Fanuc TP program (LS listing): ultrahose.ls

/PROG  ultrahose
/ATTR
COMMENT	= "19-03-20 09:29:25";
PROG_SIZE	= 0;
DEFAULT_GROUP	= 1, *, *, *, *;
/APPL
    ARC Welding Equipment: 1, *, *, *, *;
/MN
   1:  CALL HOME_ALL;
   1:  UFRAME_NUM = 1;
   1:  UTOOL_NUM = 3;
   1:  COL GUARD ADJUST 150;
   1:  PR[91] = PR[90];
   1:  PR[91,1] = PR[90,1] + -71.989;
   1:  PR[91,2] = PR[90,2] + -18.440;
   1:  PR[91,3] = PR[90,3] + 1.495;
   1:  PR[92] = PR[91];
   1:  PR[92,3] = PR[92,3] + 20;
   1:J PR[92] 10% FINE;
   1:L PR[91] R[100]mm/sec CNT100;
   1:  CALL LASER_DRAHT_START;
   1:  PR[91,1] = PR[90,1] + -66.281;
   1:  PR[91,2] = PR[90,2] + -16.361;
   1:L PR[91] R[100]mm/sec CNT100;
   1:  PR[91,1] = PR[90,1] + -66.063;
   1:  PR[91,2] = PR[90,2] + -16.303;
   1:L PR[91] R[100]mm/sec CNT100;
   1:  PR[91,1] = PR[90,1] + -66.021;
   1:  PR[91,2] = PR[90,2] + -16.273;
   1:L PR[91] R[100]mm/sec CNT100;
   1:  PR[91,1] = PR[90,1] + -61.333;
   1:  PR[91,2] = PR[90,2] + -12.339;
   1:L PR[91] R[100]mm/sec CNT100;
   1:  PR[91,1] = PR[90,1] + -61.289;
   1:  PR[91,2] = PR[90,2] + -12.295;
   1:L PR[91] R[100]mm/sec CNT100;
   1:  PR[91,1] = PR[90,1] + -61.252;
   1:  PR[91,2] = PR[90,2] + -12.242;
   1:L PR[91] R[100]mm/sec CNT100;
   1:  PR[91,1] = PR[90,1] + -58.200;
   1:  PR[91,2] = PR[90,2] + -6.959;
   1:L PR[91] R[100]mm/sec CNT100;
   1:  PR[91,1] = PR[90,1] + -57.138;
   1:  PR[91,2] = PR[90,2] + -0.935;
   1:L PR[91] R[100]mm/sec CNT100;
   1:  PR[91,1] = PR[90,1] + -57.094;
   1:  PR[91,2] = PR[90,2] + -0.772;
   1:L PR[91] R[100]mm/sec CNT100;
   1:  PR[91,1] = PR[90,1] + -58.150;
   1:  PR[91,2] = PR[90,2] + 5.213;
   1:L PR[91] R[100]mm/sec CNT100;
   1:  PR[91,1] = PR[90,1] + -58.165;
   1:  PR[91,2] = PR[90,2] + 5.381;
   1:L PR[91] R[100]mm/sec CNT100;
   1:  PR[91,1] = PR[90,1] + -61.202;
   1:  PR[91,2] = PR[90,2] + 10.640;
   1:L PR[91] R[100]mm/sec CNT100;
   1:  PR[91,1] = PR[90,1] + -61.273;
   1:  PR[91,2] = PR[90,2] + 10.794;
   1:L PR[91] R[100]mm/sec CNT100;
   1:  PR[91,1] = PR[90,1] + -65.925;
   1:  PR[91,2] = PR[90,2] + 14.697;
   1:L PR[91] R[100]mm/sec CNT100;
   1:  PR[91,1] = PR[90,1] + -66.045;
   1:  PR[91,2] = PR[90,2] + 14.817;
   1:L PR[91] R[100]mm/sec CNT100;
   1:  PR[91,1] = PR[90,1] + -71.753;
   1:  PR[91,2] = PR[90,2] + 16.895;
   1:L PR[91] R[100]mm/sec CNT100;
   1:  PR[91,1] = PR[90,1] + -71.906;
   1:  PR[91,2] = PR[90,2] + 16.966;
   1:L PR[91] R[100]mm/sec CNT100;
   1:  PR[91,1] = PR[90,1] + -77.984;
   1:L PR[91] R[100]mm/sec CNT100;
   1:  PR[91,1] = PR[90,1] + -78.152;
   1:  PR[91,2] = PR[90,2] + 16.981;
   1:L PR[91] R[100]mm/sec CNT100;
   1:  PR[91,1] = PR[90,1] + -83.860;
   1:  PR[91,2] = PR[90,2] + 14.903;
   1:L PR[91] R[100]mm/sec CNT100;
   1:  PR[91,1] = PR[90,1] + -84.078;
   1:  PR[91,2] = PR[90,2] + 14.844;
   1:L PR[91] R[100]mm/sec CNT100;
   1:  PR[91,1] = PR[90,1] + -84.120;
   1:  PR[91,2] = PR[90,2] + 14.815;
   1:L PR[91] R[100]mm/sec CNT100;
   1:  PR[91,1] = PR[90,1] + -88.808;
   1:  PR[91,2] = PR[90,2] + 10.881;
   1:L PR[91] R[100]mm/sec CNT100;
   1:  PR[91,1] = PR[90,1] + -88.852;
   1:  PR[91,2] = PR[90,2] + 10.836;
   1:L PR[91] R[100]mm/sec CNT100;
   1:  PR[91,1] = PR[90,1] + -88.889;
   1:  PR[91,2] = PR[90,2] + 10.784;
   1:L PR[91] R[100]mm/sec CNT100;
   1:  PR[91,1] = PR[90,1] + -91.941;
   1:  PR[91,2] = PR[90,2] + 5.500;
   1:L PR[91] R[100]mm/sec CNT100;
   1:  PR[91,1] = PR[90,1] + -93.003;
   1:  PR[91,2] = PR[90,2] + -0.524;
   1:L PR[91] R[100]mm/sec CNT100;
   1:  PR[91,1] = PR[90,1] + -93.047;
   1:  PR[91,2] = PR[90,2] + -0.687;
   1:L PR[91] R[100]mm/sec CNT100;
   1:  PR[91,1] = PR[90,1] + -91.991;
   1:  PR[91,2] = PR[90,2] + -6.671;
   1:L PR[91] R[100]mm/sec CNT100;
   1:  PR[91,1] = PR[90,1] + -91.977;
   1:  PR[91,2] = PR[90,2] + -6.840;
   1:L PR[91] R[100]mm/sec CNT100;
   1:  PR[91,1] = PR[90,1] + -88.939;
   1:  PR[91,2] = PR[90,2] + -12.099;
   1:L PR[91] R[100]mm/sec CNT100;
   1:  PR[91,1] = PR[90,1] + -88.868;
   1:  PR[91,2] = PR[90,2] + -12.252;
   1:L PR[91] R[100]mm/sec CNT100;
   1:  PR[91,1] = PR[90,1] + -84.216;
   1:  PR[91,2] = PR[90,2] + -16.156;
   1:L PR[91] R[100]mm/sec CNT100;
   1:  PR[91,1] = PR[90,1] + -84.097;
   1:  PR[91,2] = PR[90,2] + -16.275;
   1:L PR[91] R[100]mm/sec CNT100;
   1:  PR[91,1] = PR[90,1] + -78.388;
   1:  PR[91,2] = PR[90,2] + -18.354;
   1:L PR[91] R[100]mm/sec CNT100;
   1:  PR[91,1] = PR[90,1] + -78.236;
   1:  PR[91,2] = PR[90,2] + -18.425;
   1:L PR[91] R[100]mm/sec CNT100;
   1:  PR[91,1] = PR[90,1] + -72.157;
   1:L PR[91] R[100]mm/sec CNT100;
   1:  PR[91,1] = PR[90,1] + -71.989;
   1:  PR[91,2] = PR[90,2] + -18.440;
   1:L PR[91] R[100]mm/sec CNT100TB   .50sec,CALL END_PUD;
   1:  PR[92] = PR[91];
   1:  PR[92,3] = PR[92,3] + 20;
   1:J PR[92] 10% FINE;
   1:  PR[91,1] = PR[90,1] + -28.133;
   1:  PR[91,2] = PR[90,2] + -18.454;
   1:  PR[92] = PR[91];
   1:  PR[92,3] = PR[92,3] + 20;
   1:J PR[92] 10% FINE;
   1:L PR[91] R[100]mm/sec CNT100;
   1:  CALL LASER_DRAHT_START;
   1:  PR[91,1] = PR[90,1] + -22.027;
   1:L PR[91] R[100]mm/sec CNT100;
   1:  PR[91,1] = PR[90,1] + -16.281;
   1:  PR[91,2] = PR[90,2] + -16.361;
   1:L PR[91] R[100]mm/sec CNT100;
   1:  PR[91,1] = PR[90,1] + -16.118;
   1:  PR[91,2] = PR[90,2] + -16.318;
   1:L PR[91] R[100]mm/sec CNT100;
   1:  PR[91,1] = PR[90,1] + -11.466;
   1:  PR[91,2] = PR[90,2] + -12.414;
   1:L PR[91] R[100]mm/sec CNT100;
   1:  PR[91,1] = PR[90,1] + -11.328;
   1:  PR[91,2] = PR[90,2] + -12.317;
   1:L PR[91] R[100]mm/sec CNT100;
   1:  PR[91,1] = PR[90,1] + -8.290;
   1:  PR[91,2] = PR[90,2] + -7.058;
   1:L PR[91] R[100]mm/sec CNT100;
   1:  PR[91,1] = PR[90,1] + -8.193;
   1:  PR[91,2] = PR[90,2] + -6.919;
   1:L PR[91] R[100]mm/sec CNT100;
   1:  PR[91,1] = PR[90,1] + -7.138;
   1:  PR[91,2] = PR[90,2] + -0.935;
   1:L PR[91] R[100]mm/sec CNT100;
   1:  PR[91,1] = PR[90,1] + -7.094;
   1:  PR[91,2] = PR[90,2] + -0.772;
   1:L PR[91] R[100]mm/sec CNT100;
   1:  PR[91,1] = PR[90,1] + -8.150;
   1:  PR[91,2] = PR[90,2] + 5.213;
   1:L PR[91] R[100]mm/sec CNT100;
   1:  PR[91,1] = PR[90,1] + -8.169;
   1:  PR[91,2] = PR[90,2] + 5.437;
   1:L PR[91] R[100]mm/sec CNT100;
   1:  PR[91,1] = PR[90,1] + -8.191;
   1:  PR[91,2] = PR[90,2] + 5.484;
   1:L PR[91] R[100]mm/sec CNT100;
   1:  PR[91,1] = PR[90,1] + -11.252;
   1:  PR[91,2] = PR[90,2] + 10.784;
   1:L PR[91] R[100]mm/sec CNT100;
   1:  PR[91,1] = PR[90,1] + -11.288;
   1:  PR[91,2] = PR[90,2] + 10.836;
   1:L PR[91] R[100]mm/sec CNT100;
   1:  PR[91,1] = PR[90,1] + -11.333;
   1:  PR[91,2] = PR[90,2] + 10.881;
   1:L PR[91] R[100]mm/sec CNT100;
   1:  PR[91,1] = PR[90,1] + -16.021;
   1:  PR[91,2] = PR[90,2] + 14.815;
   1:L PR[91] R[100]mm/sec CNT100;
   1:  PR[91,1] = PR[90,1] + -16.073;
   1:  PR[91,2] = PR[90,2] + 14.851;
   1:L PR[91] R[100]mm/sec CNT100;
   1:  PR[91,1] = PR[90,1] + -16.131;
   1:  PR[91,2] = PR[90,2] + 14.878;
   1:L PR[91] R[100]mm/sec CNT100;
   1:  PR[91,1] = PR[90,1] + -21.883;
   1:  PR[91,2] = PR[90,2] + 16.973;
   1:L PR[91] R[100]mm/sec CNT100;
   1:  PR[91,1] = PR[90,1] + -21.945;
   1:  PR[91,2] = PR[90,2] + 16.989;
   1:L PR[91] R[100]mm/sec CNT100;
   1:  PR[91,1] = PR[90,1] + -22.008;
   1:  PR[91,2] = PR[90,2] + 16.995;
   1:L PR[91] R[100]mm/sec CNT100;
   1:  PR[91,1] = PR[90,1] + -28.115;
   1:L PR[91] R[100]mm/sec CNT100;
   1:  PR[91,1] = PR[90,1] + -33.860;
   1:  PR[91,2] = PR[90,2] + 14.903;
   1:L PR[91] R[100]mm/sec CNT100;
   1:  PR[91,1] = PR[90,1] + -34.023;
   1:  PR[91,2] = PR[90,2] + 14.859;
   1:L PR[91] R[100]mm/sec CNT100;
   1:  PR[91,1] = PR[90,1] + -38.675;
   1:  PR[91,2] = PR[90,2] + 10.955;
   1:L PR[91] R[100]mm/sec CNT100;
   1:  PR[91,1] = PR[90,1] + -38.813;
   1:  PR[91,2] = PR[90,2] + 10.858;
   1:L PR[91] R[100]mm/sec CNT100;
   1:  PR[91,1] = PR[90,1] + -41.851;
   1:  PR[91,2] = PR[90,2] + 5.599;
   1:L PR[91] R[100]mm/sec CNT100;
   1:  PR[91,1] = PR[90,1] + -41.948;
   1:  PR[91,2] = PR[90,2] + 5.461;
   1:L PR[91] R[100]mm/sec CNT100;
   1:  PR[91,1] = PR[90,1] + -43.004;
   1:  PR[91,2] = PR[90,2] + -0.524;
   1:L PR[91] R[100]mm/sec CNT100;
   1:  PR[91,1] = PR[90,1] + -43.047;
   1:  PR[91,2] = PR[90,2] + -0.687;
   1:L PR[91] R[100]mm/sec CNT100;
   1:  PR[91,1] = PR[90,1] + -41.991;
   1:  PR[91,2] = PR[90,2] + -6.671;
   1:L PR[91] R[100]mm/sec CNT100;
   1:  PR[91,1] = PR[90,1] + -41.972;
   1:  PR[91,2] = PR[90,2] + -6.896;
   1:L PR[91] R[100]mm/sec CNT100;
   1:  PR[91,1] = PR[90,1] + -41.950;
   1:  PR[91,2] = PR[90,2] + -6.942;
   1:L PR[91] R[100]mm/sec CNT100;
   1:  PR[91,1] = PR[90,1] + -38.889;
   1:  PR[91,2] = PR[90,2] + -12.243;
   1:L PR[91] R[100]mm/sec CNT100;
   1:  PR[91,1] = PR[90,1] + -38.853;
   1:  PR[91,2] = PR[90,2] + -12.295;
   1:L PR[91] R[100]mm/sec CNT100;
   1:  PR[91,1] = PR[90,1] + -38.808;
   1:  PR[91,2] = PR[90,2] + -12.340;
   1:L PR[91] R[100]mm/sec CNT100;
   1:  PR[91,1] = PR[90,1] + -34.120;
   1:  PR[91,2] = PR[90,2] + -16.274;
   1:L PR[91] R[100]mm/sec CNT100;
   1:  PR[91,1] = PR[90,1] + -34.068;
   1:  PR[91,2] = PR[90,2] + -16.310;
   1:L PR[91] R[100]mm/sec CNT100;
   1:  PR[91,1] = PR[90,1] + -34.010;
   1:  PR[91,2] = PR[90,2] + -16.337;
   1:L PR[91] R[100]mm/sec CNT100;
   1:  PR[91,1] = PR[90,1] + -28.258;
   1:  PR[91,2] = PR[90,2] + -18.432;
   1:L PR[91] R[100]mm/sec CNT100;
   1:  PR[91,1] = PR[90,1] + -28.197;
   1:  PR[91,2] = PR[90,2] + -18.448;
   1:L PR[91] R[100]mm/sec CNT100;
   1:  PR[91,1] = PR[90,1] + -28.133;
   1:  PR[91,2] = PR[90,2] + -18.454;
   1:L PR[91] R[100]mm/sec CNT100TB   .50sec,CALL END_PUD;
   1:  PR[92] = PR[91];
   1:  PR[92,3] = PR[92,3] + 20;
   1:J PR[92] 10% FINE;
   1:  PR[91,1] = PR[90,1] + 11.061;
   1:  PR[91,2] = PR[90,2] + -12.099;
   1:  PR[92] = PR[91];
   1:  PR[92,3] = PR[92,3] + 20;
   1:J PR[92] 10% FINE;
   1:L PR[91] R[100]mm/sec CNT100;
   1:  CALL LASER_DRAHT_START;
   1:  PR[91,1] = PR[90,1] + 11.132;
   1:  PR[91,2] = PR[90,2] + -12.252;
   1:L PR[91] R[100]mm/sec CNT100;
   1:  PR[91,1] = PR[90,1] + 15.784;
   1:  PR[91,2] = PR[90,2] + -16.156;
   1:L PR[91] R[100]mm/sec CNT100;
   1:  PR[91,1] = PR[90,1] + 15.903;
   1:  PR[91,2] = PR[90,2] + -16.275;
   1:L PR[91] R[100]mm/sec CNT100;
   1:  PR[91,1] = PR[90,1] + 21.612;
   1:  PR[91,2] = PR[90,2] + -18.354;
   1:L PR[91] R[100]mm/sec CNT100;
   1:  PR[91,1] = PR[90,1] + 21.764;
   1:  PR[91,2] = PR[90,2] + -18.425;
   1:L PR[91] R[100]mm/sec CNT100;
   1:  PR[91,1] = PR[90,1] + 27.843;
   1:L PR[91] R[100]mm/sec CNT100;
   1:  PR[91,1] = PR[90,1] + 28.011;
   1:  PR[91,2] = PR[90,2] + -18.440;
   1:L PR[91] R[100]mm/sec CNT100;
   1:  PR[91,1] = PR[90,1] + 33.719;
   1:  PR[91,2] = PR[90,2] + -16.361;
   1:L PR[91] R[100]mm/sec CNT100;
   1:  PR[91,1] = PR[90,1] + 33.937;
   1:  PR[91,2] = PR[90,2] + -16.303;
   1:L PR[91] R[100]mm/sec CNT100;
   1:  PR[91,1] = PR[90,1] + 33.979;
   1:  PR[91,2] = PR[90,2] + -16.273;
   1:L PR[91] R[100]mm/sec CNT100;
   1:  PR[91,1] = PR[90,1] + 38.667;
   1:  PR[91,2] = PR[90,2] + -12.339;
   1:L PR[91] R[100]mm/sec CNT100;
   1:  PR[91,1] = PR[90,1] + 38.711;
   1:  PR[91,2] = PR[90,2] + -12.295;
   1:L PR[91] R[100]mm/sec CNT100;
   1:  PR[91,1] = PR[90,1] + 38.748;
   1:  PR[91,2] = PR[90,2] + -12.242;
   1:L PR[91] R[100]mm/sec CNT100;
   1:  PR[91,1] = PR[90,1] + 41.800;
   1:  PR[91,2] = PR[90,2] + -6.959;
   1:L PR[91] R[100]mm/sec CNT100;
   1:  PR[91,1] = PR[90,1] + 42.862;
   1:  PR[91,2] = PR[90,2] + -0.935;
   1:L PR[91] R[100]mm/sec CNT100;
   1:  PR[91,1] = PR[90,1] + 42.906;
   1:  PR[91,2] = PR[90,2] + -0.772;
   1:L PR[91] R[100]mm/sec CNT100;
   1:  PR[91,1] = PR[90,1] + 41.850;
   1:  PR[91,2] = PR[90,2] + 5.213;
   1:L PR[91] R[100]mm/sec CNT100;
   1:  PR[91,1] = PR[90,1] + 41.835;
   1:  PR[91,2] = PR[90,2] + 5.381;
   1:L PR[91] R[100]mm/sec CNT100;
   1:  PR[91,1] = PR[90,1] + 38.798;
   1:  PR[91,2] = PR[90,2] + 10.640;
   1:L PR[91] R[100]mm/sec CNT100;
   1:  PR[91,1] = PR[90,1] + 38.727;
   1:  PR[91,2] = PR[90,2] + 10.794;
   1:L PR[91] R[100]mm/sec CNT100;
   1:  PR[91,1] = PR[90,1] + 34.075;
   1:  PR[91,2] = PR[90,2] + 14.697;
   1:L PR[91] R[100]mm/sec CNT100;
   1:  PR[91,1] = PR[90,1] + 33.956;
   1:  PR[91,2] = PR[90,2] + 14.817;
   1:L PR[91] R[100]mm/sec CNT100;
   1:  PR[91,1] = PR[90,1] + 28.247;
   1:  PR[91,2] = PR[90,2] + 16.895;
   1:L PR[91] R[100]mm/sec CNT100;
   1:  PR[91,1] = PR[90,1] + 28.094;
   1:  PR[91,2] = PR[90,2] + 16.966;
   1:L PR[91] R[100]mm/sec CNT100;
   1:  PR[91,1] = PR[90,1] + 22.016;
   1:L PR[91] R[100]mm/sec CNT100;
   1:  PR[91,1] = PR[90,1] + 21.848;
   1:  PR[91,2] = PR[90,2] + 16.981;
   1:L PR[91] R[100]mm/sec CNT100;
   1:  PR[91,1] = PR[90,1] + 16.140;
   1:  PR[91,2] = PR[90,2] + 14.903;
   1:L PR[91] R[100]mm/sec CNT100;
   1:  PR[91,1] = PR[90,1] + 15.922;
   1:  PR[91,2] = PR[90,2] + 14.844;
   1:L PR[91] R[100]mm/sec CNT100;
   1:  PR[91,1] = PR[90,1] + 15.880;
   1:  PR[91,2] = PR[90,2] + 14.815;
   1:L PR[91] R[100]mm/sec CNT100;
   1:  PR[91,1] = PR[90,1] + 11.192;
   1:  PR[91,2] = PR[90,2] + 10.881;
   1:L PR[91] R[100]mm/sec CNT100;
   1:  PR[91,1] = PR[90,1] + 11.148;
   1:  PR[91,2] = PR[90,2] + 10.836;
   1:L PR[91] R[100]mm/sec CNT100;
   1:  PR[91,1] = PR[90,1] + 11.111;
   1:  PR[91,2] = PR[90,2] + 10.784;
   1:L PR[91] R[100]mm/sec CNT100;
   1:  PR[91,1] = PR[90,1] + 8.059;
   1:  PR[91,2] = PR[90,2] + 5.500;
   1:L PR[91] R[100]mm/sec CNT100;
   1:  PR[91,1] = PR[90,1] + 6.997;
   1:  PR[91,2] = PR[90,2] + -0.524;
   1:L PR[91] R[100]mm/sec CNT100;
   1:  PR[91,1] = PR[90,1] + 6.953;
   1:  PR[91,2] = PR[90,2] + -0.687;
   1:L PR[91] R[100]mm/sec CNT100;
   1:  PR[91,1] = PR[90,1] + 8.009;
   1:  PR[91,2] = PR[90,2] + -6.671;
   1:L PR[91] R[100]mm/sec CNT100;
   1:  PR[91,1] = PR[90,1] + 8.023;
   1:  PR[91,2] = PR[90,2] + -6.840;
   1:L PR[91] R[100]mm/sec CNT100;
   1:  PR[91,1] = PR[90,1] + 11.061;
   1:  PR[91,2] = PR[90,2] + -12.099;
   1:L PR[91] R[100]mm/sec CNT100TB   .50sec,CALL END_PUD;
   1:  PR[92] = PR[91];
   1:  PR[92,3] = PR[92,3] + 20;
   1:J PR[92] 10% FINE;
   1:  PR[91,1] = PR[90,1] + 91.852;
   1:  PR[91,2] = PR[90,2] + -6.823;
   1:  PR[92] = PR[91];
   1:  PR[92,3] = PR[92,3] + 20;
   1:J PR[92] 10% FINE;
   1:L PR[91] R[100]mm/sec CNT100;
   1:  CALL LASER_DRAHT_START;
   1:  PR[91,1] = PR[90,1] + 92.913;
   1:  PR[91,2] = PR[90,2] + -0.811;
   1:L PR[91] R[100]mm/sec CNT100;
   1:  PR[91,1] = PR[90,1] + 91.850;
   1:  PR[91,2] = PR[90,2] + 5.213;
   1:L PR[91] R[100]mm/sec CNT100;
   1:  PR[91,1] = PR[90,1] + 91.831;
   1:  PR[91,2] = PR[90,2] + 5.437;
   1:L PR[91] R[100]mm/sec CNT100;
   1:  PR[91,1] = PR[90,1] + 91.809;
   1:  PR[91,2] = PR[90,2] + 5.483;
   1:L PR[91] R[100]mm/sec CNT100;
   1:  PR[91,1] = PR[90,1] + 88.757;
   1:  PR[91,2] = PR[90,2] + 10.768;
   1:L PR[91] R[100]mm/sec CNT100;
   1:  PR[91,1] = PR[90,1] + 84.075;
   1:  PR[91,2] = PR[90,2] + 14.697;
   1:L PR[91] R[100]mm/sec CNT100;
   1:  PR[91,1] = PR[90,1] + 83.956;
   1:  PR[91,2] = PR[90,2] + 14.816;
   1:L PR[91] R[100]mm/sec CNT100;
   1:  PR[91,1] = PR[90,1] + 78.248;
   1:  PR[91,2] = PR[90,2] + 16.895;
   1:L PR[91] R[100]mm/sec CNT100;
   1:  PR[91,1] = PR[90,1] + 78.043;
   1:  PR[91,2] = PR[90,2] + 16.990;
   1:L PR[91] R[100]mm/sec CNT100;
   1:  PR[91,1] = PR[90,1] + 77.993;
   1:  PR[91,2] = PR[90,2] + 16.995;
   1:L PR[91] R[100]mm/sec CNT100;
   1:  PR[91,1] = PR[90,1] + 71.867;
   1:L PR[91] R[100]mm/sec CNT100;
   1:  PR[91,1] = PR[90,1] + 71.803;
   1:  PR[91,2] = PR[90,2] + 16.989;
   1:L PR[91] R[100]mm/sec CNT100;
   1:  PR[91,1] = PR[90,1] + 71.742;
   1:  PR[91,2] = PR[90,2] + 16.973;
   1:L PR[91] R[100]mm/sec CNT100;
   1:  PR[91,1] = PR[90,1] + 65.990;
   1:  PR[91,2] = PR[90,2] + 14.878;
   1:L PR[91] R[100]mm/sec CNT100;
   1:  PR[91,1] = PR[90,1] + 65.932;
   1:  PR[91,2] = PR[90,2] + 14.851;
   1:L PR[91] R[100]mm/sec CNT100;
   1:  PR[91,1] = PR[90,1] + 65.880;
   1:  PR[91,2] = PR[90,2] + 14.815;
   1:L PR[91] R[100]mm/sec CNT100;
   1:  PR[91,1] = PR[90,1] + 61.192;
   1:  PR[91,2] = PR[90,2] + 10.881;
   1:L PR[91] R[100]mm/sec CNT100;
   1:  PR[91,1] = PR[90,1] + 61.148;
   1:  PR[91,2] = PR[90,2] + 10.836;
   1:L PR[91] R[100]mm/sec CNT100;
   1:  PR[91,1] = PR[90,1] + 61.111;
   1:  PR[91,2] = PR[90,2] + 10.784;
   1:L PR[91] R[100]mm/sec CNT100;
   1:  PR[91,1] = PR[90,1] + 58.050;
   1:  PR[91,2] = PR[90,2] + 5.484;
   1:L PR[91] R[100]mm/sec CNT100;
   1:  PR[91,1] = PR[90,1] + 58.023;
   1:  PR[91,2] = PR[90,2] + 5.426;
   1:L PR[91] R[100]mm/sec CNT100;
   1:  PR[91,1] = PR[90,1] + 58.007;
   1:  PR[91,2] = PR[90,2] + 5.365;
   1:L PR[91] R[100]mm/sec CNT100;
   1:  PR[91,1] = PR[90,1] + 56.946;
   1:  PR[91,2] = PR[90,2] + -0.648;
   1:L PR[91] R[100]mm/sec CNT100;
   1:  PR[91,1] = PR[90,1] + 58.009;
   1:  PR[91,2] = PR[90,2] + -6.671;
   1:L PR[91] R[100]mm/sec CNT100;
   1:  PR[91,1] = PR[90,1] + 58.028;
   1:  PR[91,2] = PR[90,2] + -6.896;
   1:L PR[91] R[100]mm/sec CNT100;
   1:  PR[91,1] = PR[90,1] + 58.050;
   1:  PR[91,2] = PR[90,2] + -6.942;
   1:L PR[91] R[100]mm/sec CNT100;
   1:  PR[91,1] = PR[90,1] + 61.102;
   1:  PR[91,2] = PR[90,2] + -12.227;
   1:L PR[91] R[100]mm/sec CNT100;
   1:  PR[91,1] = PR[90,1] + 65.784;
   1:  PR[91,2] = PR[90,2] + -16.156;
   1:L PR[91] R[100]mm/sec CNT100;
   1:  PR[91,1] = PR[90,1] + 65.903;
   1:  PR[91,2] = PR[90,2] + -16.275;
   1:L PR[91] R[100]mm/sec CNT100;
   1:  PR[91,1] = PR[90,1] + 71.611;
   1:  PR[91,2] = PR[90,2] + -18.354;
   1:L PR[91] R[100]mm/sec CNT100;
   1:  PR[91,1] = PR[90,1] + 71.816;
   1:  PR[91,2] = PR[90,2] + -18.449;
   1:L PR[91] R[100]mm/sec CNT100;
   1:  PR[91,1] = PR[90,1] + 71.866;
   1:  PR[91,2] = PR[90,2] + -18.454;
   1:L PR[91] R[100]mm/sec CNT100;
   1:  PR[91,1] = PR[90,1] + 77.992;
   1:L PR[91] R[100]mm/sec CNT100;
   1:  PR[91,1] = PR[90,1] + 78.055;
   1:  PR[91,2] = PR[90,2] + -18.448;
   1:L PR[91] R[100]mm/sec CNT100;
   1:  PR[91,1] = PR[90,1] + 78.116;
   1:  PR[91,2] = PR[90,2] + -18.432;
   1:L PR[91] R[100]mm/sec CNT100;
   1:  PR[91,1] = PR[90,1] + 83.869;
   1:  PR[91,2] = PR[90,2] + -16.337;
   1:L PR[91] R[100]mm/sec CNT100;
   1:  PR[91,1] = PR[90,1] + 83.927;
   1:  PR[91,2] = PR[90,2] + -16.310;
   1:L PR[91] R[100]mm/sec CNT100;
   1:  PR[91,1] = PR[90,1] + 83.979;
   1:  PR[91,2] = PR[90,2] + -16.274;
   1:L PR[91] R[100]mm/sec CNT100;
   1:  PR[91,1] = PR[90,1] + 88.667;
   1:  PR[91,2] = PR[90,2] + -12.340;
   1:L PR[91] R[100]mm/sec CNT100;
   1:  PR[91,1] = PR[90,1] + 88.711;
   1:  PR[91,2] = PR[90,2] + -12.295;
   1:L PR[91] R[100]mm/sec CNT100;
   1:  PR[91,1] = PR[90,1] + 88.748;
   1:  PR[91,2] = PR[90,2] + -12.242;
   1:L PR[91] R[100]mm/sec CNT100;
   1:  PR[91,1] = PR[90,1] + 91.809;
   1:  PR[91,2] = PR[90,2] + -6.943;
   1:L PR[91] R[100]mm/sec CNT100;
   1:  PR[91,1] = PR[90,1] + 91.836;
   1:  PR[91,2] = PR[90,2] + -6.885;
   1:L PR[91] R[100]mm/sec CNT100;
   1:  PR[91,1] = PR[90,1] + 91.852;
   1:  PR[91,2] = PR[90,2] + -6.823;
   1:L PR[91] R[100]mm/sec CNT100TB   .50sec,CALL END_PUD;
   1:  PR[92] = PR[91];
   1:  PR[92,3] = PR[92,3] + 20;
   1:J PR[92] 10% FINE;
   1:  PR[91] = PR[90];
   1:  PR[91,1] = PR[90,1] + -66.602;
   1:  PR[91,2] = PR[90,2] + -16.557;
   1:  PR[91,3] = PR[90,3] + 2.795;
   1:  PR[92] = PR[91];
   1:  PR[92,3] = PR[92,3] + 20;
   1:J PR[92] 10% FINE;
   1:L PR[91] R[100]mm/sec CNT100;
   1:  CALL LASER_DRAHT_START;
   1:  PR[91,1] = PR[90,1] + -66.074;
   1:  PR[91,2] = PR[90,2] + -16.310;
   1:L PR[91] R[100]mm/sec CNT100;
   1:  PR[91,1] = PR[90,1] + -65.522;
   1:  PR[91,2] = PR[90,2] + -15.924;
   1:L PR[91] R[100]mm/sec CNT100;
   1:  PR[91,1] = PR[90,1] + -61.763;
   1:  PR[91,2] = PR[90,2] + -12.770;
   1:L PR[91] R[100]mm/sec CNT100;
   1:  PR[91,1] = PR[90,1] + -61.289;
   1:  PR[91,2] = PR[90,2] + -12.295;
   1:L PR[91] R[100]mm/sec CNT100;
   1:  PR[91,1] = PR[90,1] + -60.902;
   1:  PR[91,2] = PR[90,2] + -11.743;
   1:L PR[91] R[100]mm/sec CNT100;
   1:  PR[91,1] = PR[90,1] + -58.448;
   1:  PR[91,2] = PR[90,2] + -7.493;
   1:L PR[91] R[100]mm/sec CNT100;
   1:  PR[91,1] = PR[90,1] + -58.201;
   1:  PR[91,2] = PR[90,2] + -6.965;
   1:L PR[91] R[100]mm/sec CNT100;
   1:  PR[91,1] = PR[90,1] + -57.348;
   1:  PR[91,2] = PR[90,2] + -2.130;
   1:L PR[91] R[100]mm/sec CNT100;
   1:  PR[91,1] = PR[90,1] + -57.129;
   1:  PR[91,2] = PR[90,2] + -1.311;
   1:L PR[91] R[100]mm/sec CNT100;
   1:  PR[91,1] = PR[90,1] + -57.086;
   1:  PR[91,2] = PR[90,2] + -0.818;
   1:L PR[91] R[100]mm/sec CNT100;
   1:  PR[91,1] = PR[90,1] + -57.939;
   1:  PR[91,2] = PR[90,2] + 4.017;
   1:L PR[91] R[100]mm/sec CNT100;
   1:  PR[91,1] = PR[90,1] + -58.013;
   1:  PR[91,2] = PR[90,2] + 4.860;
   1:L PR[91] R[100]mm/sec CNT100;
   1:  PR[91,1] = PR[90,1] + -58.141;
   1:  PR[91,2] = PR[90,2] + 5.341;
   1:L PR[91] R[100]mm/sec CNT100;
   1:  PR[91,1] = PR[90,1] + -60.595;
   1:  PR[91,2] = PR[90,2] + 9.589;
   1:L PR[91] R[100]mm/sec CNT100;
   1:  PR[91,1] = PR[90,1] + -60.953;
   1:  PR[91,2] = PR[90,2] + 10.357;
   1:L PR[91] R[100]mm/sec CNT100;
   1:  PR[91,1] = PR[90,1] + -61.239;
   1:  PR[91,2] = PR[90,2] + 10.765;
   1:L PR[91] R[100]mm/sec CNT100;
   1:  PR[91,1] = PR[90,1] + -64.997;
   1:  PR[91,2] = PR[90,2] + 13.919;
   1:L PR[91] R[100]mm/sec CNT100;
   1:  PR[91,1] = PR[90,1] + -65.595;
   1:  PR[91,2] = PR[90,2] + 14.516;
   1:L PR[91] R[100]mm/sec CNT100;
   1:  PR[91,1] = PR[90,1] + -66.003;
   1:  PR[91,2] = PR[90,2] + 14.802;
   1:L PR[91] R[100]mm/sec CNT100;
   1:  PR[91,1] = PR[90,1] + -70.614;
   1:  PR[91,2] = PR[90,2] + 16.481;
   1:L PR[91] R[100]mm/sec CNT100;
   1:  PR[91,1] = PR[90,1] + -71.381;
   1:  PR[91,2] = PR[90,2] + 16.838;
   1:L PR[91] R[100]mm/sec CNT100;
   1:  PR[91,1] = PR[90,1] + -71.861;
   1:  PR[91,2] = PR[90,2] + 16.967;
   1:L PR[91] R[100]mm/sec CNT100;
   1:  PR[91,1] = PR[90,1] + -76.772;
   1:L PR[91] R[100]mm/sec CNT100;
   1:  PR[91,1] = PR[90,1] + -77.615;
   1:  PR[91,2] = PR[90,2] + 17.040;
   1:L PR[91] R[100]mm/sec CNT100;
   1:  PR[91,1] = PR[90,1] + -78.109;
   1:  PR[91,2] = PR[90,2] + 16.997;
   1:L PR[91] R[100]mm/sec CNT100;
   1:  PR[91,1] = PR[90,1] + -82.720;
   1:  PR[91,2] = PR[90,2] + 15.318;
   1:L PR[91] R[100]mm/sec CNT100;
   1:  PR[91,1] = PR[90,1] + -83.539;
   1:  PR[91,2] = PR[90,2] + 15.098;
   1:L PR[91] R[100]mm/sec CNT100;
   1:  PR[91,1] = PR[90,1] + -84.067;
   1:  PR[91,2] = PR[90,2] + 14.852;
   1:L PR[91] R[100]mm/sec CNT100;
   1:  PR[91,1] = PR[90,1] + -84.619;
   1:  PR[91,2] = PR[90,2] + 14.465;
   1:L PR[91] R[100]mm/sec CNT100;
   1:  PR[91,1] = PR[90,1] + -88.378;
   1:  PR[91,2] = PR[90,2] + 11.311;
   1:L PR[91] R[100]mm/sec CNT100;
   1:  PR[91,1] = PR[90,1] + -88.852;
   1:  PR[91,2] = PR[90,2] + 10.837;
   1:L PR[91] R[100]mm/sec CNT100;
   1:  PR[91,1] = PR[90,1] + -89.239;
   1:  PR[91,2] = PR[90,2] + 10.284;
   1:L PR[91] R[100]mm/sec CNT100;
   1:  PR[91,1] = PR[90,1] + -91.693;
   1:  PR[91,2] = PR[90,2] + 6.035;
   1:L PR[91] R[100]mm/sec CNT100;
   1:  PR[91,1] = PR[90,1] + -91.940;
   1:  PR[91,2] = PR[90,2] + 5.506;
   1:L PR[91] R[100]mm/sec CNT100;
   1:  PR[91,1] = PR[90,1] + -92.793;
   1:  PR[91,2] = PR[90,2] + 0.671;
   1:L PR[91] R[100]mm/sec CNT100;
   1:  PR[91,1] = PR[90,1] + -93.012;
   1:  PR[91,2] = PR[90,2] + -0.148;
   1:L PR[91] R[100]mm/sec CNT100;
   1:  PR[91,1] = PR[90,1] + -93.055;
   1:  PR[91,2] = PR[90,2] + -0.641;
   1:L PR[91] R[100]mm/sec CNT100;
   1:  PR[91,1] = PR[90,1] + -92.202;
   1:  PR[91,2] = PR[90,2] + -5.476;
   1:L PR[91] R[100]mm/sec CNT100;
   1:  PR[91,1] = PR[90,1] + -92.129;
   1:  PR[91,2] = PR[90,2] + -6.319;
   1:L PR[91] R[100]mm/sec CNT100;
   1:  PR[91,1] = PR[90,1] + -92.000;
   1:  PR[91,2] = PR[90,2] + -6.800;
   1:L PR[91] R[100]mm/sec CNT100;
   1:  PR[91,1] = PR[90,1] + -89.546;
   1:  PR[91,2] = PR[90,2] + -11.048;
   1:L PR[91] R[100]mm/sec CNT100;
   1:  PR[91,1] = PR[90,1] + -89.188;
   1:  PR[91,2] = PR[90,2] + -11.816;
   1:L PR[91] R[100]mm/sec CNT100;
   1:  PR[91,1] = PR[90,1] + -88.902;
   1:  PR[91,2] = PR[90,2] + -12.224;
   1:L PR[91] R[100]mm/sec CNT100;
   1:  PR[91,1] = PR[90,1] + -85.144;
   1:  PR[91,2] = PR[90,2] + -15.377;
   1:L PR[91] R[100]mm/sec CNT100;
   1:  PR[91,1] = PR[90,1] + -84.546;
   1:  PR[91,2] = PR[90,2] + -15.975;
   1:L PR[91] R[100]mm/sec CNT100;
   1:  PR[91,1] = PR[90,1] + -84.138;
   1:  PR[91,2] = PR[90,2] + -16.261;
   1:L PR[91] R[100]mm/sec CNT100;
   1:  PR[91,1] = PR[90,1] + -79.527;
   1:  PR[91,2] = PR[90,2] + -17.940;
   1:L PR[91] R[100]mm/sec CNT100;
   1:  PR[91,1] = PR[90,1] + -78.760;
   1:  PR[91,2] = PR[90,2] + -18.297;
   1:L PR[91] R[100]mm/sec CNT100;
   1:  PR[91,1] = PR[90,1] + -78.280;
   1:  PR[91,2] = PR[90,2] + -18.426;
   1:L PR[91] R[100]mm/sec CNT100;
   1:  PR[91,1] = PR[90,1] + -73.369;
   1:L PR[91] R[100]mm/sec CNT100;
   1:  PR[91,1] = PR[90,1] + -72.526;
   1:  PR[91,2] = PR[90,2] + -18.499;
   1:L PR[91] R[100]mm/sec CNT100;
   1:  PR[91,1] = PR[90,1] + -72.032;
   1:  PR[91,2] = PR[90,2] + -18.456;
   1:L PR[91] R[100]mm/sec CNT100;
   1:  PR[91,1] = PR[90,1] + -67.421;
   1:  PR[91,2] = PR[90,2] + -16.776;
   1:L PR[91] R[100]mm/sec CNT100;
   1:  PR[91,1] = PR[90,1] + -66.602;
   1:  PR[91,2] = PR[90,2] + -16.557;
   1:L PR[91] R[100]mm/sec CNT100TB   .50sec,CALL END_PUD;
   1:  PR[92] = PR[91];
   1:  PR[92,3] = PR[92,3] + 20;
   1:J PR[92] 10% FINE;
   1:  PR[91,1] = PR[90,1] + -7.129;
   1:  PR[91,2] = PR[90,2] + -1.311;
   1:  PR[92] = PR[91];
   1:  PR[92,3] = PR[92,3] + 20;
   1:J PR[92] 10% FINE;
   1:L PR[91] R[100]mm/sec CNT100;
   1:  CALL LASER_DRAHT_START;
   1:  PR[91,1] = PR[90,1] + -7.086;
   1:  PR[91,2] = PR[90,2] + -0.818;
   1:L PR[91] R[100]mm/sec CNT100;
   1:  PR[91,1] = PR[90,1] + -7.939;
   1:  PR[91,2] = PR[90,2] + 4.017;
   1:L PR[91] R[100]mm/sec CNT100;
   1:  PR[91,1] = PR[90,1] + -8.013;
   1:  PR[91,2] = PR[90,2] + 4.860;
   1:L PR[91] R[100]mm/sec CNT100;
   1:  PR[91,1] = PR[90,1] + -8.164;
   1:  PR[91,2] = PR[90,2] + 5.425;
   1:L PR[91] R[100]mm/sec CNT100;
   1:  PR[91,1] = PR[90,1] + -8.448;
   1:  PR[91,2] = PR[90,2] + 6.035;
   1:L PR[91] R[100]mm/sec CNT100;
   1:  PR[91,1] = PR[90,1] + -10.902;
   1:  PR[91,2] = PR[90,2] + 10.284;
   1:L PR[91] R[100]mm/sec CNT100;
   1:  PR[91,1] = PR[90,1] + -11.288;
   1:  PR[91,2] = PR[90,2] + 10.835;
   1:L PR[91] R[100]mm/sec CNT100;
   1:  PR[91,1] = PR[90,1] + -11.763;
   1:  PR[91,2] = PR[90,2] + 11.311;
   1:L PR[91] R[100]mm/sec CNT100;
   1:  PR[91,1] = PR[90,1] + -15.522;
   1:  PR[91,2] = PR[90,2] + 14.465;
   1:L PR[91] R[100]mm/sec CNT100;
   1:  PR[91,1] = PR[90,1] + -16.073;
   1:  PR[91,2] = PR[90,2] + 14.851;
   1:L PR[91] R[100]mm/sec CNT100;
   1:  PR[91,1] = PR[90,1] + -16.682;
   1:  PR[91,2] = PR[90,2] + 15.135;
   1:L PR[91] R[100]mm/sec CNT100;
   1:  PR[91,1] = PR[90,1] + -21.295;
   1:  PR[91,2] = PR[90,2] + 16.815;
   1:L PR[91] R[100]mm/sec CNT100;
   1:  PR[91,1] = PR[90,1] + -21.944;
   1:  PR[91,2] = PR[90,2] + 16.989;
   1:L PR[91] R[100]mm/sec CNT100;
   1:  PR[91,1] = PR[90,1] + -22.615;
   1:  PR[91,2] = PR[90,2] + 17.048;
   1:L PR[91] R[100]mm/sec CNT100;
   1:  PR[91,1] = PR[90,1] + -27.526;
   1:L PR[91] R[100]mm/sec CNT100;
   1:  PR[91,1] = PR[90,1] + -28.109;
   1:  PR[91,2] = PR[90,2] + 16.997;
   1:L PR[91] R[100]mm/sec CNT100;
   1:  PR[91,1] = PR[90,1] + -32.720;
   1:  PR[91,2] = PR[90,2] + 15.318;
   1:L PR[91] R[100]mm/sec CNT100;
   1:  PR[91,1] = PR[90,1] + -33.538;
   1:  PR[91,2] = PR[90,2] + 15.098;
   1:L PR[91] R[100]mm/sec CNT100;
   1:  PR[91,1] = PR[90,1] + -33.988;
   1:  PR[91,2] = PR[90,2] + 14.888;
   1:L PR[91] R[100]mm/sec CNT100;
   1:  PR[91,1] = PR[90,1] + -37.746;
   1:  PR[91,2] = PR[90,2] + 11.735;
   1:L PR[91] R[100]mm/sec CNT100;
   1:  PR[91,1] = PR[90,1] + -38.439;
   1:  PR[91,2] = PR[90,2] + 11.249;
   1:L PR[91] R[100]mm/sec CNT100;
   1:  PR[91,1] = PR[90,1] + -38.791;
   1:  PR[91,2] = PR[90,2] + 10.898;
   1:L PR[91] R[100]mm/sec CNT100;
   1:  PR[91,1] = PR[90,1] + -41.245;
   1:  PR[91,2] = PR[90,2] + 6.649;
   1:L PR[91] R[100]mm/sec CNT100;
   1:  PR[91,1] = PR[90,1] + -41.730;
   1:  PR[91,2] = PR[90,2] + 5.956;
   1:L PR[91] R[100]mm/sec CNT100;
   1:  PR[91,1] = PR[90,1] + -41.940;
   1:  PR[91,2] = PR[90,2] + 5.505;
   1:L PR[91] R[100]mm/sec CNT100;
   1:  PR[91,1] = PR[90,1] + -42.793;
   1:  PR[91,2] = PR[90,2] + 0.670;
   1:L PR[91] R[100]mm/sec CNT100;
   1:  PR[91,1] = PR[90,1] + -43.012;
   1:  PR[91,2] = PR[90,2] + -0.148;
   1:L PR[91] R[100]mm/sec CNT100;
   1:  PR[91,1] = PR[90,1] + -43.055;
   1:  PR[91,2] = PR[90,2] + -0.641;
   1:L PR[91] R[100]mm/sec CNT100;
   1:  PR[91,1] = PR[90,1] + -42.202;
   1:  PR[91,2] = PR[90,2] + -5.476;
   1:L PR[91] R[100]mm/sec CNT100;
   1:  PR[91,1] = PR[90,1] + -42.129;
   1:  PR[91,2] = PR[90,2] + -6.319;
   1:L PR[91] R[100]mm/sec CNT100;
   1:  PR[91,1] = PR[90,1] + -41.977;
   1:  PR[91,2] = PR[90,2] + -6.884;
   1:L PR[91] R[100]mm/sec CNT100;
   1:  PR[91,1] = PR[90,1] + -41.693;
   1:  PR[91,2] = PR[90,2] + -7.493;
   1:L PR[91] R[100]mm/sec CNT100;
   1:  PR[91,1] = PR[90,1] + -39.239;
   1:  PR[91,2] = PR[90,2] + -11.743;
   1:L PR[91] R[100]mm/sec CNT100;
   1:  PR[91,1] = PR[90,1] + -38.853;
   1:  PR[91,2] = PR[90,2] + -12.294;
   1:L PR[91] R[100]mm/sec CNT100;
   1:  PR[91,1] = PR[90,1] + -38.378;
   1:  PR[91,2] = PR[90,2] + -12.770;
   1:L PR[91] R[100]mm/sec CNT100;
   1:  PR[91,1] = PR[90,1] + -34.619;
   1:  PR[91,2] = PR[90,2] + -15.924;
   1:L PR[91] R[100]mm/sec CNT100;
   1:  PR[91,1] = PR[90,1] + -34.069;
   1:  PR[91,2] = PR[90,2] + -16.310;
   1:L PR[91] R[100]mm/sec CNT100;
   1:  PR[91,1] = PR[90,1] + -33.459;
   1:  PR[91,2] = PR[90,2] + -16.594;
   1:L PR[91] R[100]mm/sec CNT100;
   1:  PR[91,1] = PR[90,1] + -28.846;
   1:  PR[91,2] = PR[90,2] + -18.274;
   1:L PR[91] R[100]mm/sec CNT100;
   1:  PR[91,1] = PR[90,1] + -28.197;
   1:  PR[91,2] = PR[90,2] + -18.448;
   1:L PR[91] R[100]mm/sec CNT100;
   1:  PR[91,1] = PR[90,1] + -27.527;
   1:  PR[91,2] = PR[90,2] + -18.507;
   1:L PR[91] R[100]mm/sec CNT100;
   1:  PR[91,1] = PR[90,1] + -22.615;
   1:L PR[91] R[100]mm/sec CNT100;
   1:  PR[91,1] = PR[90,1] + -22.033;
   1:  PR[91,2] = PR[90,2] + -18.456;
   1:L PR[91] R[100]mm/sec CNT100;
   1:  PR[91,1] = PR[90,1] + -17.421;
   1:  PR[91,2] = PR[90,2] + -16.777;
   1:L PR[91] R[100]mm/sec CNT100;
   1:  PR[91,1] = PR[90,1] + -16.603;
   1:  PR[91,2] = PR[90,2] + -16.557;
   1:L PR[91] R[100]mm/sec CNT100;
   1:  PR[91,1] = PR[90,1] + -16.153;
   1:  PR[91,2] = PR[90,2] + -16.347;
   1:L PR[91] R[100]mm/sec CNT100;
   1:  PR[91,1] = PR[90,1] + -12.395;
   1:  PR[91,2] = PR[90,2] + -13.194;
   1:L PR[91] R[100]mm/sec CNT100;
   1:  PR[91,1] = PR[90,1] + -11.702;
   1:  PR[91,2] = PR[90,2] + -12.708;
   1:L PR[91] R[100]mm/sec CNT100;
   1:  PR[91,1] = PR[90,1] + -11.350;
   1:  PR[91,2] = PR[90,2] + -12.356;
   1:L PR[91] R[100]mm/sec CNT100;
   1:  PR[91,1] = PR[90,1] + -8.897;
   1:  PR[91,2] = PR[90,2] + -8.108;
   1:L PR[91] R[100]mm/sec CNT100;
   1:  PR[91,1] = PR[90,1] + -8.411;
   1:  PR[91,2] = PR[90,2] + -7.415;
   1:L PR[91] R[100]mm/sec CNT100;
   1:  PR[91,1] = PR[90,1] + -8.201;
   1:  PR[91,2] = PR[90,2] + -6.964;
   1:L PR[91] R[100]mm/sec CNT100;
   1:  PR[91,1] = PR[90,1] + -7.348;
   1:  PR[91,2] = PR[90,2] + -2.129;
   1:L PR[91] R[100]mm/sec CNT100;
   1:  PR[91,1] = PR[90,1] + -7.129;
   1:  PR[91,2] = PR[90,2] + -1.311;
   1:L PR[91] R[100]mm/sec CNT100TB   .50sec,CALL END_PUD;
   1:  PR[92] = PR[91];
   1:  PR[92,3] = PR[92,3] + 20;
   1:J PR[92] 10% FINE;
   1:  PR[91,1] = PR[90,1] + 11.148;
   1:  PR[91,2] = PR[90,2] + 10.837;
   1:  PR[92] = PR[91];
   1:  PR[92,3] = PR[92,3] + 20;
   1:J PR[92] 10% FINE;
   1:L PR[91] R[100]mm/sec CNT100;
   1:  CALL LASER_DRAHT_START;
   1:  PR[91,1] = PR[90,1] + 10.761;
   1:  PR[91,2] = PR[90,2] + 10.284;
   1:L PR[91] R[100]mm/sec CNT100;
   1:  PR[91,1] = PR[90,1] + 8.307;
   1:  PR[91,2] = PR[90,2] + 6.035;
   1:L PR[91] R[100]mm/sec CNT100;
   1:  PR[91,1] = PR[90,1] + 8.060;
   1:  PR[91,2] = PR[90,2] + 5.506;
   1:L PR[91] R[100]mm/sec CNT100;
   1:  PR[91,1] = PR[90,1] + 7.207;
   1:  PR[91,2] = PR[90,2] + 0.671;
   1:L PR[91] R[100]mm/sec CNT100;
   1:  PR[91,1] = PR[90,1] + 6.988;
   1:  PR[91,2] = PR[90,2] + -0.148;
   1:L PR[91] R[100]mm/sec CNT100;
   1:  PR[91,1] = PR[90,1] + 6.945;
   1:  PR[91,2] = PR[90,2] + -0.641;
   1:L PR[91] R[100]mm/sec CNT100;
   1:  PR[91,1] = PR[90,1] + 7.798;
   1:  PR[91,2] = PR[90,2] + -5.476;
   1:L PR[91] R[100]mm/sec CNT100;
   1:  PR[91,1] = PR[90,1] + 7.871;
   1:  PR[91,2] = PR[90,2] + -6.319;
   1:L PR[91] R[100]mm/sec CNT100;
   1:  PR[91,1] = PR[90,1] + 8.000;
   1:  PR[91,2] = PR[90,2] + -6.800;
   1:L PR[91] R[100]mm/sec CNT100;
   1:  PR[91,1] = PR[90,1] + 10.454;
   1:  PR[91,2] = PR[90,2] + -11.048;
   1:L PR[91] R[100]mm/sec CNT100;
   1:  PR[91,1] = PR[90,1] + 10.812;
   1:  PR[91,2] = PR[90,2] + -11.816;
   1:L PR[91] R[100]mm/sec CNT100;
   1:  PR[91,1] = PR[90,1] + 11.098;
   1:  PR[91,2] = PR[90,2] + -12.224;
   1:L PR[91] R[100]mm/sec CNT100;
   1:  PR[91,1] = PR[90,1] + 14.855;
   1:  PR[91,2] = PR[90,2] + -15.377;
   1:L PR[91] R[100]mm/sec CNT100;
   1:  PR[91,1] = PR[90,1] + 15.454;
   1:  PR[91,2] = PR[90,2] + -15.975;
   1:L PR[91] R[100]mm/sec CNT100;
   1:  PR[91,1] = PR[90,1] + 15.862;
   1:  PR[91,2] = PR[90,2] + -16.261;
   1:L PR[91] R[100]mm/sec CNT100;
   1:  PR[91,1] = PR[90,1] + 20.473;
   1:  PR[91,2] = PR[90,2] + -17.940;
   1:L PR[91] R[100]mm/sec CNT100;
   1:  PR[91,1] = PR[90,1] + 21.240;
   1:  PR[91,2] = PR[90,2] + -18.297;
   1:L PR[91] R[100]mm/sec CNT100;
   1:  PR[91,1] = PR[90,1] + 21.720;
   1:  PR[91,2] = PR[90,2] + -18.426;
   1:L PR[91] R[100]mm/sec CNT100;
   1:  PR[91,1] = PR[90,1] + 26.631;
   1:L PR[91] R[100]mm/sec CNT100;
   1:  PR[91,1] = PR[90,1] + 27.474;
   1:  PR[91,2] = PR[90,2] + -18.499;
   1:L PR[91] R[100]mm/sec CNT100;
   1:  PR[91,1] = PR[90,1] + 27.968;
   1:  PR[91,2] = PR[90,2] + -18.456;
   1:L PR[91] R[100]mm/sec CNT100;
   1:  PR[91,1] = PR[90,1] + 32.579;
   1:  PR[91,2] = PR[90,2] + -16.776;
   1:L PR[91] R[100]mm/sec CNT100;
   1:  PR[91,1] = PR[90,1] + 33.398;
   1:  PR[91,2] = PR[90,2] + -16.557;
   1:L PR[91] R[100]mm/sec CNT100;
   1:  PR[91,1] = PR[90,1] + 33.926;
   1:  PR[91,2] = PR[90,2] + -16.310;
   1:L PR[91] R[100]mm/sec CNT100;
   1:  PR[91,1] = PR[90,1] + 34.478;
   1:  PR[91,2] = PR[90,2] + -15.924;
   1:L PR[91] R[100]mm/sec CNT100;
   1:  PR[91,1] = PR[90,1] + 38.237;
   1:  PR[91,2] = PR[90,2] + -12.770;
   1:L PR[91] R[100]mm/sec CNT100;
   1:  PR[91,1] = PR[90,1] + 38.711;
   1:  PR[91,2] = PR[90,2] + -12.295;
   1:L PR[91] R[100]mm/sec CNT100;
   1:  PR[91,1] = PR[90,1] + 39.098;
   1:  PR[91,2] = PR[90,2] + -11.743;
   1:L PR[91] R[100]mm/sec CNT100;
   1:  PR[91,1] = PR[90,1] + 41.552;
   1:  PR[91,2] = PR[90,2] + -7.493;
   1:L PR[91] R[100]mm/sec CNT100;
   1:  PR[91,1] = PR[90,1] + 41.799;
   1:  PR[91,2] = PR[90,2] + -6.965;
   1:L PR[91] R[100]mm/sec CNT100;
   1:  PR[91,1] = PR[90,1] + 42.652;
   1:  PR[91,2] = PR[90,2] + -2.130;
   1:L PR[91] R[100]mm/sec CNT100;
   1:  PR[91,1] = PR[90,1] + 42.871;
   1:  PR[91,2] = PR[90,2] + -1.311;
   1:L PR[91] R[100]mm/sec CNT100;
   1:  PR[91,1] = PR[90,1] + 42.914;
   1:  PR[91,2] = PR[90,2] + -0.818;
   1:L PR[91] R[100]mm/sec CNT100;
   1:  PR[91,1] = PR[90,1] + 42.061;
   1:  PR[91,2] = PR[90,2] + 4.017;
   1:L PR[91] R[100]mm/sec CNT100;
   1:  PR[91,1] = PR[90,1] + 41.987;
   1:  PR[91,2] = PR[90,2] + 4.860;
   1:L PR[91] R[100]mm/sec CNT100;
   1:  PR[91,1] = PR[90,1] + 41.859;
   1:  PR[91,2] = PR[90,2] + 5.341;
   1:L PR[91] R[100]mm/sec CNT100;
   1:  PR[91,1] = PR[90,1] + 39.405;
   1:  PR[91,2] = PR[90,2] + 9.589;
   1:L PR[91] R[100]mm/sec CNT100;
   1:  PR[91,1] = PR[90,1] + 39.047;
   1:  PR[91,2] = PR[90,2] + 10.357;
   1:L PR[91] R[100]mm/sec CNT100;
   1:  PR[91,1] = PR[90,1] + 38.761;
   1:  PR[91,2] = PR[90,2] + 10.765;
   1:L PR[91] R[100]mm/sec CNT100;
   1:  PR[91,1] = PR[90,1] + 35.003;
   1:  PR[91,2] = PR[90,2] + 13.919;
   1:L PR[91] R[100]mm/sec CNT100;
   1:  PR[91,1] = PR[90,1] + 34.405;
   1:  PR[91,2] = PR[90,2] + 14.516;
   1:L PR[91] R[100]mm/sec CNT100;
   1:  PR[91,1] = PR[90,1] + 33.997;
   1:  PR[91,2] = PR[90,2] + 14.802;
   1:L PR[91] R[100]mm/sec CNT100;
   1:  PR[91,1] = PR[90,1] + 29.386;
   1:  PR[91,2] = PR[90,2] + 16.481;
   1:L PR[91] R[100]mm/sec CNT100;
   1:  PR[91,1] = PR[90,1] + 28.619;
   1:  PR[91,2] = PR[90,2] + 16.838;
   1:L PR[91] R[100]mm/sec CNT100;
   1:  PR[91,1] = PR[90,1] + 28.139;
   1:  PR[91,2] = PR[90,2] + 16.967;
   1:L PR[91] R[100]mm/sec CNT100;
   1:  PR[91,1] = PR[90,1] + 23.228;
   1:L PR[91] R[100]mm/sec CNT100;
   1:  PR[91,1] = PR[90,1] + 22.385;
   1:  PR[91,2] = PR[90,2] + 17.040;
   1:L PR[91] R[100]mm/sec CNT100;
   1:  PR[91,1] = PR[90,1] + 21.891;
   1:  PR[91,2] = PR[90,2] + 16.997;
   1:L PR[91] R[100]mm/sec CNT100;
   1:  PR[91,1] = PR[90,1] + 17.280;
   1:  PR[91,2] = PR[90,2] + 15.318;
   1:L PR[91] R[100]mm/sec CNT100;
   1:  PR[91,1] = PR[90,1] + 16.461;
   1:  PR[91,2] = PR[90,2] + 15.098;
   1:L PR[91] R[100]mm/sec CNT100;
   1:  PR[91,1] = PR[90,1] + 15.933;
   1:  PR[91,2] = PR[90,2] + 14.852;
   1:L PR[91] R[100]mm/sec CNT100;
   1:  PR[91,1] = PR[90,1] + 15.381;
   1:  PR[91,2] = PR[90,2] + 14.465;
   1:L PR[91] R[100]mm/sec CNT100;
   1:  PR[91,1] = PR[90,1] + 11.622;
   1:  PR[91,2] = PR[90,2] + 11.311;
   1:L PR[91] R[100]mm/sec CNT100;
   1:  PR[91,1] = PR[90,1] + 11.148;
   1:  PR[91,2] = PR[90,2] + 10.837;
   1:L PR[91] R[100]mm/sec CNT100TB   .50sec,CALL END_PUD;
   1:  PR[92] = PR[91];
   1:  PR[92,3] = PR[92,3] + 20;
   1:J PR[92] 10% FINE;
   1:  PR[91,1] = PR[90,1] + 88.236;
   1:  PR[91,2] = PR[90,2] + -12.771;
   1:  PR[92] = PR[91];
   1:  PR[92,3] = PR[92,3] + 20;
   1:J PR[92] 10% FINE;
   1:L PR[91] R[100]mm/sec CNT100;
   1:  CALL LASER_DRAHT_START;
   1:  PR[91,1] = PR[90,1] + 88.710;
   1:  PR[91,2] = PR[90,2] + -12.296;
   1:L PR[91] R[100]mm/sec CNT100;
   1:  PR[91,1] = PR[90,1] + 89.097;
   1:  PR[91,2] = PR[90,2] + -11.744;
   1:L PR[91] R[100]mm/sec CNT100;
   1:  PR[91,1] = PR[90,1] + 91.552;
   1:  PR[91,2] = PR[90,2] + -7.494;
   1:L PR[91] R[100]mm/sec CNT100;
   1:  PR[91,1] = PR[90,1] + 91.836;
   1:  PR[91,2] = PR[90,2] + -6.885;
   1:L PR[91] R[100]mm/sec CNT100;
   1:  PR[91,1] = PR[90,1] + 92.010;
   1:  PR[91,2] = PR[90,2] + -6.234;
   1:L PR[91] R[100]mm/sec CNT100;
   1:  PR[91,1] = PR[90,1] + 92.863;
   1:  PR[91,2] = PR[90,2] + -1.398;
   1:L PR[91] R[100]mm/sec CNT100;
   1:  PR[91,1] = PR[90,1] + 92.914;
   1:  PR[91,2] = PR[90,2] + -0.818;
   1:L PR[91] R[100]mm/sec CNT100;
   1:  PR[91,1] = PR[90,1] + 92.061;
   1:  PR[91,2] = PR[90,2] + 4.017;
   1:L PR[91] R[100]mm/sec CNT100;
   1:  PR[91,1] = PR[90,1] + 91.987;
   1:  PR[91,2] = PR[90,2] + 4.860;
   1:L PR[91] R[100]mm/sec CNT100;
   1:  PR[91,1] = PR[90,1] + 91.836;
   1:  PR[91,2] = PR[90,2] + 5.426;
   1:L PR[91] R[100]mm/sec CNT100;
   1:  PR[91,1] = PR[90,1] + 91.552;
   1:  PR[91,2] = PR[90,2] + 6.035;
   1:L PR[91] R[100]mm/sec CNT100;
   1:  PR[91,1] = PR[90,1] + 89.098;
   1:  PR[91,2] = PR[90,2] + 10.284;
   1:L PR[91] R[100]mm/sec CNT100;
   1:  PR[91,1] = PR[90,1] + 88.762;
   1:  PR[91,2] = PR[90,2] + 10.764;
   1:L PR[91] R[100]mm/sec CNT100;
   1:  PR[91,1] = PR[90,1] + 85.004;
   1:  PR[91,2] = PR[90,2] + 13.918;
   1:L PR[91] R[100]mm/sec CNT100;
   1:  PR[91,1] = PR[90,1] + 84.406;
   1:  PR[91,2] = PR[90,2] + 14.515;
   1:L PR[91] R[100]mm/sec CNT100;
   1:  PR[91,1] = PR[90,1] + 83.999;
   1:  PR[91,2] = PR[90,2] + 14.801;
   1:L PR[91] R[100]mm/sec CNT100;
   1:  PR[91,1] = PR[90,1] + 79.387;
   1:  PR[91,2] = PR[90,2] + 16.480;
   1:L PR[91] R[100]mm/sec CNT100;
   1:  PR[91,1] = PR[90,1] + 78.621;
   1:  PR[91,2] = PR[90,2] + 16.838;
   1:L PR[91] R[100]mm/sec CNT100;
   1:  PR[91,1] = PR[90,1] + 78.056;
   1:  PR[91,2] = PR[90,2] + 16.989;
   1:L PR[91] R[100]mm/sec CNT100;
   1:  PR[91,1] = PR[90,1] + 77.387;
   1:  PR[91,2] = PR[90,2] + 17.048;
   1:L PR[91] R[100]mm/sec CNT100;
   1:  PR[91,1] = PR[90,1] + 72.475;
   1:L PR[91] R[100]mm/sec CNT100;
   1:  PR[91,1] = PR[90,1] + 71.805;
   1:  PR[91,2] = PR[90,2] + 16.990;
   1:L PR[91] R[100]mm/sec CNT100;
   1:  PR[91,1] = PR[90,1] + 71.155;
   1:  PR[91,2] = PR[90,2] + 16.816;
   1:L PR[91] R[100]mm/sec CNT100;
   1:  PR[91,1] = PR[90,1] + 66.543;
   1:  PR[91,2] = PR[90,2] + 15.136;
   1:L PR[91] R[100]mm/sec CNT100;
   1:  PR[91,1] = PR[90,1] + 65.934;
   1:  PR[91,2] = PR[90,2] + 14.852;
   1:L PR[91] R[100]mm/sec CNT100;
   1:  PR[91,1] = PR[90,1] + 65.382;
   1:  PR[91,2] = PR[90,2] + 14.466;
   1:L PR[91] R[100]mm/sec CNT100;
   1:  PR[91,1] = PR[90,1] + 61.623;
   1:  PR[91,2] = PR[90,2] + 11.312;
   1:L PR[91] R[100]mm/sec CNT100;
   1:  PR[91,1] = PR[90,1] + 61.148;
   1:  PR[91,2] = PR[90,2] + 10.837;
   1:L PR[91] R[100]mm/sec CNT100;
   1:  PR[91,1] = PR[90,1] + 60.761;
   1:  PR[91,2] = PR[90,2] + 10.285;
   1:L PR[91] R[100]mm/sec CNT100;
   1:  PR[91,1] = PR[90,1] + 58.307;
   1:  PR[91,2] = PR[90,2] + 6.035;
   1:L PR[91] R[100]mm/sec CNT100;
   1:  PR[91,1] = PR[90,1] + 58.023;
   1:  PR[91,2] = PR[90,2] + 5.426;
   1:L PR[91] R[100]mm/sec CNT100;
   1:  PR[91,1] = PR[90,1] + 57.849;
   1:  PR[91,2] = PR[90,2] + 4.775;
   1:L PR[91] R[100]mm/sec CNT100;
   1:  PR[91,1] = PR[90,1] + 56.995;
   1:  PR[91,2] = PR[90,2] + -0.061;
   1:L PR[91] R[100]mm/sec CNT100;
   1:  PR[91,1] = PR[90,1] + 56.945;
   1:  PR[91,2] = PR[90,2] + -0.641;
   1:L PR[91] R[100]mm/sec CNT100;
   1:  PR[91,1] = PR[90,1] + 57.798;
   1:  PR[91,2] = PR[90,2] + -5.476;
   1:L PR[91] R[100]mm/sec CNT100;
   1:  PR[91,1] = PR[90,1] + 57.871;
   1:  PR[91,2] = PR[90,2] + -6.319;
   1:L PR[91] R[100]mm/sec CNT100;
   1:  PR[91,1] = PR[90,1] + 58.023;
   1:  PR[91,2] = PR[90,2] + -6.885;
   1:L PR[91] R[100]mm/sec CNT100;
   1:  PR[91,1] = PR[90,1] + 58.307;
   1:  PR[91,2] = PR[90,2] + -7.493;
   1:L PR[91] R[100]mm/sec CNT100;
   1:  PR[91,1] = PR[90,1] + 60.761;
   1:  PR[91,2] = PR[90,2] + -11.743;
   1:L PR[91] R[100]mm/sec CNT100;
   1:  PR[91,1] = PR[90,1] + 61.097;
   1:  PR[91,2] = PR[90,2] + -12.223;
   1:L PR[91] R[100]mm/sec CNT100;
   1:  PR[91,1] = PR[90,1] + 64.855;
   1:  PR[91,2] = PR[90,2] + -15.376;
   1:L PR[91] R[100]mm/sec CNT100;
   1:  PR[91,1] = PR[90,1] + 65.453;
   1:  PR[91,2] = PR[90,2] + -15.974;
   1:L PR[91] R[100]mm/sec CNT100;
   1:  PR[91,1] = PR[90,1] + 65.860;
   1:  PR[91,2] = PR[90,2] + -16.260;
   1:L PR[91] R[100]mm/sec CNT100;
   1:  PR[91,1] = PR[90,1] + 70.471;
   1:  PR[91,2] = PR[90,2] + -17.939;
   1:L PR[91] R[100]mm/sec CNT100;
   1:  PR[91,1] = PR[90,1] + 71.238;
   1:  PR[91,2] = PR[90,2] + -18.296;
   1:L PR[91] R[100]mm/sec CNT100;
   1:  PR[91,1] = PR[90,1] + 71.803;
   1:  PR[91,2] = PR[90,2] + -18.448;
   1:L PR[91] R[100]mm/sec CNT100;
   1:  PR[91,1] = PR[90,1] + 72.472;
   1:  PR[91,2] = PR[90,2] + -18.507;
   1:L PR[91] R[100]mm/sec CNT100;
   1:  PR[91,1] = PR[90,1] + 77.384;
   1:L PR[91] R[100]mm/sec CNT100;
   1:  PR[91,1] = PR[90,1] + 78.054;
   1:  PR[91,2] = PR[90,2] + -18.448;
   1:L PR[91] R[100]mm/sec CNT100;
   1:  PR[91,1] = PR[90,1] + 78.703;
   1:  PR[91,2] = PR[90,2] + -18.274;
   1:L PR[91] R[100]mm/sec CNT100;
   1:  PR[91,1] = PR[90,1] + 83.316;
   1:  PR[91,2] = PR[90,2] + -16.595;
   1:L PR[91] R[100]mm/sec CNT100;
   1:  PR[91,1] = PR[90,1] + 83.925;
   1:  PR[91,2] = PR[90,2] + -16.311;
   1:L PR[91] R[100]mm/sec CNT100;
   1:  PR[91,1] = PR[90,1] + 84.477;
   1:  PR[91,2] = PR[90,2] + -15.925;
   1:L PR[91] R[100]mm/sec CNT100;
   1:  PR[91,1] = PR[90,1] + 88.236;
   1:  PR[91,2] = PR[90,2] + -12.771;
   1:L PR[91] R[100]mm/sec CNT100TB   .50sec,CALL END_PUD;
   1:  PR[92] = PR[91];
   1:  PR[92,3] = PR[92,3] + 20;
   1:J PR[92] 10% FINE;
   1:  PR[91] = PR[90];
   1:  PR[91,1] = PR[90,1] + -58.687;
   1:  PR[91,2] = PR[90,2] + -8.006;
   1:  PR[91,3] = PR[90,3] + 4.095;
   1:  PR[92] = PR[91];
   1:  PR[92,3] = PR[92,3] + 20;
   1:J PR[92] 10% FINE;
   1:L PR[91] R[100]mm/sec CNT100;
   1:  CALL LASER_DRAHT_START;
   1:  PR[91,1] = PR[90,1] + -58.201;
   1:  PR[91,2] = PR[90,2] + -6.964;
   1:L PR[91] R[100]mm/sec CNT100;
   1:  PR[91,1] = PR[90,1] + -57.544;
   1:  PR[91,2] = PR[90,2] + -3.242;
   1:L PR[91] R[100]mm/sec CNT100;
   1:  PR[91,1] = PR[90,1] + -57.178;
   1:  PR[91,2] = PR[90,2] + -1.875;
   1:L PR[91] R[100]mm/sec CNT100;
   1:  PR[91,1] = PR[90,1] + -57.086;
   1:  PR[91,2] = PR[90,2] + -0.818;
   1:L PR[91] R[100]mm/sec CNT100;
   1:  PR[91,1] = PR[90,1] + -57.743;
   1:  PR[91,2] = PR[90,2] + 2.905;
   1:L PR[91] R[100]mm/sec CNT100;
   1:  PR[91,1] = PR[90,1] + -57.866;
   1:  PR[91,2] = PR[90,2] + 4.312;
   1:L PR[91] R[100]mm/sec CNT100;
   1:  PR[91,1] = PR[90,1] + -58.141;
   1:  PR[91,2] = PR[90,2] + 5.341;
   1:L PR[91] R[100]mm/sec CNT100;
   1:  PR[91,1] = PR[90,1] + -60.031;
   1:  PR[91,2] = PR[90,2] + 8.612;
   1:L PR[91] R[100]mm/sec CNT100;
   1:  PR[91,1] = PR[90,1] + -60.628;
   1:  PR[91,2] = PR[90,2] + 9.893;
   1:L PR[91] R[100]mm/sec CNT100;
   1:  PR[91,1] = PR[90,1] + -61.240;
   1:  PR[91,2] = PR[90,2] + 10.766;
   1:L PR[91] R[100]mm/sec CNT100;
   1:  PR[91,1] = PR[90,1] + -64.133;
   1:  PR[91,2] = PR[90,2] + 13.194;
   1:L PR[91] R[100]mm/sec CNT100;
   1:  PR[91,1] = PR[90,1] + -65.131;
   1:  PR[91,2] = PR[90,2] + 14.192;
   1:L PR[91] R[100]mm/sec CNT100;
   1:  PR[91,1] = PR[90,1] + -66.005;
   1:  PR[91,2] = PR[90,2] + 14.803;
   1:L PR[91] R[100]mm/sec CNT100;
   1:  PR[91,1] = PR[90,1] + -69.555;
   1:  PR[91,2] = PR[90,2] + 16.096;
   1:L PR[91] R[100]mm/sec CNT100;
   1:  PR[91,1] = PR[90,1] + -70.835;
   1:  PR[91,2] = PR[90,2] + 16.692;
   1:L PR[91] R[100]mm/sec CNT100;
   1:  PR[91,1] = PR[90,1] + -71.863;
   1:  PR[91,2] = PR[90,2] + 16.967;
   1:L PR[91] R[100]mm/sec CNT100;
   1:  PR[91,1] = PR[90,1] + -75.644;
   1:L PR[91] R[100]mm/sec CNT100;
   1:  PR[91,1] = PR[90,1] + -77.052;
   1:  PR[91,2] = PR[90,2] + 17.090;
   1:L PR[91] R[100]mm/sec CNT100;
   1:  PR[91,1] = PR[90,1] + -78.110;
   1:  PR[91,2] = PR[90,2] + 16.997;
   1:L PR[91] R[100]mm/sec CNT100;
   1:  PR[91,1] = PR[90,1] + -81.661;
   1:  PR[91,2] = PR[90,2] + 15.704;
   1:L PR[91] R[100]mm/sec CNT100;
   1:  PR[91,1] = PR[90,1] + -83.026;
   1:  PR[91,2] = PR[90,2] + 15.337;
   1:L PR[91] R[100]mm/sec CNT100;
   1:  PR[91,1] = PR[90,1] + -84.067;
   1:  PR[91,2] = PR[90,2] + 14.852;
   1:L PR[91] R[100]mm/sec CNT100;
   1:  PR[91,1] = PR[90,1] + -85.083;
   1:  PR[91,2] = PR[90,2] + 14.140;
   1:L PR[91] R[100]mm/sec CNT100;
   1:  PR[91,1] = PR[90,1] + -87.978;
   1:  PR[91,2] = PR[90,2] + 11.711;
   1:L PR[91] R[100]mm/sec CNT100;
   1:  PR[91,1] = PR[90,1] + -88.852;
   1:  PR[91,2] = PR[90,2] + 10.837;
   1:L PR[91] R[100]mm/sec CNT100;
   1:  PR[91,1] = PR[90,1] + -89.564;
   1:  PR[91,2] = PR[90,2] + 9.820;
   1:L PR[91] R[100]mm/sec CNT100;
   1:  PR[91,1] = PR[90,1] + -91.454;
   1:  PR[91,2] = PR[90,2] + 6.547;
   1:L PR[91] R[100]mm/sec CNT100;
   1:  PR[91,1] = PR[90,1] + -91.940;
   1:  PR[91,2] = PR[90,2] + 5.505;
   1:L PR[91] R[100]mm/sec CNT100;
   1:  PR[91,1] = PR[90,1] + -92.597;
   1:  PR[91,2] = PR[90,2] + 1.783;
   1:L PR[91] R[100]mm/sec CNT100;
   1:  PR[91,1] = PR[90,1] + -92.963;
   1:  PR[91,2] = PR[90,2] + 0.416;
   1:L PR[91] R[100]mm/sec CNT100;
   1:  PR[91,1] = PR[90,1] + -93.055;
   1:  PR[91,2] = PR[90,2] + -0.641;
   1:L PR[91] R[100]mm/sec CNT100;
   1:  PR[91,1] = PR[90,1] + -92.398;
   1:  PR[91,2] = PR[90,2] + -4.364;
   1:L PR[91] R[100]mm/sec CNT100;
   1:  PR[91,1] = PR[90,1] + -92.275;
   1:  PR[91,2] = PR[90,2] + -5.771;
   1:L PR[91] R[100]mm/sec CNT100;
   1:  PR[91,1] = PR[90,1] + -92.000;
   1:  PR[91,2] = PR[90,2] + -6.800;
   1:L PR[91] R[100]mm/sec CNT100;
   1:  PR[91,1] = PR[90,1] + -90.111;
   1:  PR[91,2] = PR[90,2] + -10.071;
   1:L PR[91] R[100]mm/sec CNT100;
   1:  PR[91,1] = PR[90,1] + -89.513;
   1:  PR[91,2] = PR[90,2] + -11.352;
   1:L PR[91] R[100]mm/sec CNT100;
   1:  PR[91,1] = PR[90,1] + -88.901;
   1:  PR[91,2] = PR[90,2] + -12.225;
   1:L PR[91] R[100]mm/sec CNT100;
   1:  PR[91,1] = PR[90,1] + -86.008;
   1:  PR[91,2] = PR[90,2] + -14.653;
   1:L PR[91] R[100]mm/sec CNT100;
   1:  PR[91,1] = PR[90,1] + -85.010;
   1:  PR[91,2] = PR[90,2] + -15.651;
   1:L PR[91] R[100]mm/sec CNT100;
   1:  PR[91,1] = PR[90,1] + -84.137;
   1:  PR[91,2] = PR[90,2] + -16.262;
   1:L PR[91] R[100]mm/sec CNT100;
   1:  PR[91,1] = PR[90,1] + -80.586;
   1:  PR[91,2] = PR[90,2] + -17.555;
   1:L PR[91] R[100]mm/sec CNT100;
   1:  PR[91,1] = PR[90,1] + -79.307;
   1:  PR[91,2] = PR[90,2] + -18.151;
   1:L PR[91] R[100]mm/sec CNT100;
   1:  PR[91,1] = PR[90,1] + -78.278;
   1:  PR[91,2] = PR[90,2] + -18.426;
   1:L PR[91] R[100]mm/sec CNT100;
   1:  PR[91,1] = PR[90,1] + -74.497;
   1:L PR[91] R[100]mm/sec CNT100;
   1:  PR[91,1] = PR[90,1] + -73.090;
   1:  PR[91,2] = PR[90,2] + -18.549;
   1:L PR[91] R[100]mm/sec CNT100;
   1:  PR[91,1] = PR[90,1] + -72.031;
   1:  PR[91,2] = PR[90,2] + -18.456;
   1:L PR[91] R[100]mm/sec CNT100;
   1:  PR[91,1] = PR[90,1] + -68.481;
   1:  PR[91,2] = PR[90,2] + -17.163;
   1:L PR[91] R[100]mm/sec CNT100;
   1:  PR[91,1] = PR[90,1] + -67.115;
   1:  PR[91,2] = PR[90,2] + -16.796;
   1:L PR[91] R[100]mm/sec CNT100;
   1:  PR[91,1] = PR[90,1] + -66.074;
   1:  PR[91,2] = PR[90,2] + -16.311;
   1:L PR[91] R[100]mm/sec CNT100;
   1:  PR[91,1] = PR[90,1] + -65.058;
   1:  PR[91,2] = PR[90,2] + -15.599;
   1:L PR[91] R[100]mm/sec CNT100;
   1:  PR[91,1] = PR[90,1] + -62.163;
   1:  PR[91,2] = PR[90,2] + -13.170;
   1:L PR[91] R[100]mm/sec CNT100;
   1:  PR[91,1] = PR[90,1] + -61.289;
   1:  PR[91,2] = PR[90,2] + -12.296;
   1:L PR[91] R[100]mm/sec CNT100;
   1:  PR[91,1] = PR[90,1] + -60.577;
   1:  PR[91,2] = PR[90,2] + -11.278;
   1:L PR[91] R[100]mm/sec CNT100;
   1:  PR[91,1] = PR[90,1] + -58.687;
   1:  PR[91,2] = PR[90,2] + -8.006;
   1:L PR[91] R[100]mm/sec CNT100TB   .50sec,CALL END_PUD;
   1:  PR[92] = PR[91];
   1:  PR[92,3] = PR[92,3] + 20;
   1:J PR[92] 10% FINE;
   1:  PR[91,1] = PR[90,1] + -41.940;
   1:  PR[91,2] = PR[90,2] + 5.504;
   1:  PR[92] = PR[91];
   1:  PR[92,3] = PR[92,3] + 20;
   1:J PR[92] 10% FINE;
   1:L PR[91] R[100]mm/sec CNT100;
   1:  CALL LASER_DRAHT_START;
   1:  PR[91,1] = PR[90,1] + -42.597;
   1:  PR[91,2] = PR[90,2] + 1.781;
   1:L PR[91] R[100]mm/sec CNT100;
   1:  PR[91,1] = PR[90,1] + -42.963;
   1:  PR[91,2] = PR[90,2] + 0.416;
   1:L PR[91] R[100]mm/sec CNT100;
   1:  PR[91,1] = PR[90,1] + -43.055;
   1:  PR[91,2] = PR[90,2] + -0.641;
   1:L PR[91] R[100]mm/sec CNT100;
   1:  PR[91,1] = PR[90,1] + -42.398;
   1:  PR[91,2] = PR[90,2] + -4.364;
   1:L PR[91] R[100]mm/sec CNT100;
   1:  PR[91,1] = PR[90,1] + -42.275;
   1:  PR[91,2] = PR[90,2] + -5.771;
   1:L PR[91] R[100]mm/sec CNT100;
   1:  PR[91,1] = PR[90,1] + -41.978;
   1:  PR[91,2] = PR[90,2] + -6.883;
   1:L PR[91] R[100]mm/sec CNT100;
   1:  PR[91,1] = PR[90,1] + -41.454;
   1:  PR[91,2] = PR[90,2] + -8.006;
   1:L PR[91] R[100]mm/sec CNT100;
   1:  PR[91,1] = PR[90,1] + -39.564;
   1:  PR[91,2] = PR[90,2] + -11.279;
   1:L PR[91] R[100]mm/sec CNT100;
   1:  PR[91,1] = PR[90,1] + -38.854;
   1:  PR[91,2] = PR[90,2] + -12.293;
   1:L PR[91] R[100]mm/sec CNT100;
   1:  PR[91,1] = PR[90,1] + -37.978;
   1:  PR[91,2] = PR[90,2] + -13.170;
   1:L PR[91] R[100]mm/sec CNT100;
   1:  PR[91,1] = PR[90,1] + -35.083;
   1:  PR[91,2] = PR[90,2] + -15.599;
   1:L PR[91] R[100]mm/sec CNT100;
   1:  PR[91,1] = PR[90,1] + -34.069;
   1:  PR[91,2] = PR[90,2] + -16.310;
   1:L PR[91] R[100]mm/sec CNT100;
   1:  PR[91,1] = PR[90,1] + -32.946;
   1:  PR[91,2] = PR[90,2] + -16.834;
   1:L PR[91] R[100]mm/sec CNT100;
   1:  PR[91,1] = PR[90,1] + -29.394;
   1:  PR[91,2] = PR[90,2] + -18.127;
   1:L PR[91] R[100]mm/sec CNT100;
   1:  PR[91,1] = PR[90,1] + -28.197;
   1:  PR[91,2] = PR[90,2] + -18.448;
   1:L PR[91] R[100]mm/sec CNT100;
   1:  PR[91,1] = PR[90,1] + -26.962;
   1:  PR[91,2] = PR[90,2] + -18.556;
   1:L PR[91] R[100]mm/sec CNT100;
   1:  PR[91,1] = PR[90,1] + -23.180;
   1:L PR[91] R[100]mm/sec CNT100;
   1:  PR[91,1] = PR[90,1] + -22.033;
   1:  PR[91,2] = PR[90,2] + -18.456;
   1:L PR[91] R[100]mm/sec CNT100;
   1:  PR[91,1] = PR[90,1] + -18.482;
   1:  PR[91,2] = PR[90,2] + -17.163;
   1:L PR[91] R[100]mm/sec CNT100;
   1:  PR[91,1] = PR[90,1] + -17.116;
   1:  PR[91,2] = PR[90,2] + -16.797;
   1:L PR[91] R[100]mm/sec CNT100;
   1:  PR[91,1] = PR[90,1] + -16.152;
   1:  PR[91,2] = PR[90,2] + -16.347;
   1:L PR[91] R[100]mm/sec CNT100;
   1:  PR[91,1] = PR[90,1] + -13.259;
   1:  PR[91,2] = PR[90,2] + -13.919;
   1:L PR[91] R[100]mm/sec CNT100;
   1:  PR[91,1] = PR[90,1] + -12.102;
   1:  PR[91,2] = PR[90,2] + -13.109;
   1:L PR[91] R[100]mm/sec CNT100;
   1:  PR[91,1] = PR[90,1] + -11.350;
   1:  PR[91,2] = PR[90,2] + -12.356;
   1:L PR[91] R[100]mm/sec CNT100;
   1:  PR[91,1] = PR[90,1] + -9.460;
   1:  PR[91,2] = PR[90,2] + -9.085;
   1:L PR[91] R[100]mm/sec CNT100;
   1:  PR[91,1] = PR[90,1] + -8.650;
   1:  PR[91,2] = PR[90,2] + -7.927;
   1:L PR[91] R[100]mm/sec CNT100;
   1:  PR[91,1] = PR[90,1] + -8.201;
   1:  PR[91,2] = PR[90,2] + -6.963;
   1:L PR[91] R[100]mm/sec CNT100;
   1:  PR[91,1] = PR[90,1] + -7.544;
   1:  PR[91,2] = PR[90,2] + -3.240;
   1:L PR[91] R[100]mm/sec CNT100;
   1:  PR[91,1] = PR[90,1] + -7.178;
   1:  PR[91,2] = PR[90,2] + -1.875;
   1:L PR[91] R[100]mm/sec CNT100;
   1:  PR[91,1] = PR[90,1] + -7.086;
   1:  PR[91,2] = PR[90,2] + -0.818;
   1:L PR[91] R[100]mm/sec CNT100;
   1:  PR[91,1] = PR[90,1] + -7.743;
   1:  PR[91,2] = PR[90,2] + 2.905;
   1:L PR[91] R[100]mm/sec CNT100;
   1:  PR[91,1] = PR[90,1] + -7.866;
   1:  PR[91,2] = PR[90,2] + 4.312;
   1:L PR[91] R[100]mm/sec CNT100;
   1:  PR[91,1] = PR[90,1] + -8.163;
   1:  PR[91,2] = PR[90,2] + 5.424;
   1:L PR[91] R[100]mm/sec CNT100;
   1:  PR[91,1] = PR[90,1] + -8.687;
   1:  PR[91,2] = PR[90,2] + 6.547;
   1:L PR[91] R[100]mm/sec CNT100;
   1:  PR[91,1] = PR[90,1] + -10.577;
   1:  PR[91,2] = PR[90,2] + 9.820;
   1:L PR[91] R[100]mm/sec CNT100;
   1:  PR[91,1] = PR[90,1] + -11.287;
   1:  PR[91,2] = PR[90,2] + 10.835;
   1:L PR[91] R[100]mm/sec CNT100;
   1:  PR[91,1] = PR[90,1] + -12.163;
   1:  PR[91,2] = PR[90,2] + 11.711;
   1:L PR[91] R[100]mm/sec CNT100;
   1:  PR[91,1] = PR[90,1] + -15.058;
   1:  PR[91,2] = PR[90,2] + 14.140;
   1:L PR[91] R[100]mm/sec CNT100;
   1:  PR[91,1] = PR[90,1] + -16.072;
   1:  PR[91,2] = PR[90,2] + 14.851;
   1:L PR[91] R[100]mm/sec CNT100;
   1:  PR[91,1] = PR[90,1] + -17.195;
   1:  PR[91,2] = PR[90,2] + 15.375;
   1:L PR[91] R[100]mm/sec CNT100;
   1:  PR[91,1] = PR[90,1] + -20.747;
   1:  PR[91,2] = PR[90,2] + 16.668;
   1:L PR[91] R[100]mm/sec CNT100;
   1:  PR[91,1] = PR[90,1] + -21.944;
   1:  PR[91,2] = PR[90,2] + 16.989;
   1:L PR[91] R[100]mm/sec CNT100;
   1:  PR[91,1] = PR[90,1] + -23.179;
   1:  PR[91,2] = PR[90,2] + 17.097;
   1:L PR[91] R[100]mm/sec CNT100;
   1:  PR[91,1] = PR[90,1] + -26.961;
   1:L PR[91] R[100]mm/sec CNT100;
   1:  PR[91,1] = PR[90,1] + -28.109;
   1:  PR[91,2] = PR[90,2] + 16.997;
   1:L PR[91] R[100]mm/sec CNT100;
   1:  PR[91,1] = PR[90,1] + -31.659;
   1:  PR[91,2] = PR[90,2] + 15.704;
   1:L PR[91] R[100]mm/sec CNT100;
   1:  PR[91,1] = PR[90,1] + -33.025;
   1:  PR[91,2] = PR[90,2] + 15.338;
   1:L PR[91] R[100]mm/sec CNT100;
   1:  PR[91,1] = PR[90,1] + -33.989;
   1:  PR[91,2] = PR[90,2] + 14.888;
   1:L PR[91] R[100]mm/sec CNT100;
   1:  PR[91,1] = PR[90,1] + -36.882;
   1:  PR[91,2] = PR[90,2] + 12.460;
   1:L PR[91] R[100]mm/sec CNT100;
   1:  PR[91,1] = PR[90,1] + -38.039;
   1:  PR[91,2] = PR[90,2] + 11.650;
   1:L PR[91] R[100]mm/sec CNT100;
   1:  PR[91,1] = PR[90,1] + -38.792;
   1:  PR[91,2] = PR[90,2] + 10.897;
   1:L PR[91] R[100]mm/sec CNT100;
   1:  PR[91,1] = PR[90,1] + -40.681;
   1:  PR[91,2] = PR[90,2] + 7.626;
   1:L PR[91] R[100]mm/sec CNT100;
   1:  PR[91,1] = PR[90,1] + -41.491;
   1:  PR[91,2] = PR[90,2] + 6.469;
   1:L PR[91] R[100]mm/sec CNT100;
   1:  PR[91,1] = PR[90,1] + -41.940;
   1:  PR[91,2] = PR[90,2] + 5.504;
   1:L PR[91] R[100]mm/sec CNT100TB   .50sec,CALL END_PUD;
   1:  PR[92] = PR[91];
   1:  PR[92,3] = PR[92,3] + 20;
   1:J PR[92] 10% FINE;
   1:  PR[91,1] = PR[90,1] + 28.137;
   1:  PR[91,2] = PR[90,2] + 16.967;
   1:  PR[92] = PR[91];
   1:  PR[92,3] = PR[92,3] + 20;
   1:J PR[92] 10% FINE;
   1:L PR[91] R[100]mm/sec CNT100;
   1:  CALL LASER_DRAHT_START;
   1:  PR[91,1] = PR[90,1] + 24.356;
   1:L PR[91] R[100]mm/sec CNT100;
   1:  PR[91,1] = PR[90,1] + 22.948;
   1:  PR[91,2] = PR[90,2] + 17.090;
   1:L PR[91] R[100]mm/sec CNT100;
   1:  PR[91,1] = PR[90,1] + 21.890;
   1:  PR[91,2] = PR[90,2] + 16.997;
   1:L PR[91] R[100]mm/sec CNT100;
   1:  PR[91,1] = PR[90,1] + 18.340;
   1:  PR[91,2] = PR[90,2] + 15.704;
   1:L PR[91] R[100]mm/sec CNT100;
   1:  PR[91,1] = PR[90,1] + 16.974;
   1:  PR[91,2] = PR[90,2] + 15.337;
   1:L PR[91] R[100]mm/sec CNT100;
   1:  PR[91,1] = PR[90,1] + 15.933;
   1:  PR[91,2] = PR[90,2] + 14.852;
   1:L PR[91] R[100]mm/sec CNT100;
   1:  PR[91,1] = PR[90,1] + 14.917;
   1:  PR[91,2] = PR[90,2] + 14.140;
   1:L PR[91] R[100]mm/sec CNT100;
   1:  PR[91,1] = PR[90,1] + 12.022;
   1:  PR[91,2] = PR[90,2] + 11.711;
   1:L PR[91] R[100]mm/sec CNT100;
   1:  PR[91,1] = PR[90,1] + 11.148;
   1:  PR[91,2] = PR[90,2] + 10.837;
   1:L PR[91] R[100]mm/sec CNT100;
   1:  PR[91,1] = PR[90,1] + 10.436;
   1:  PR[91,2] = PR[90,2] + 9.820;
   1:L PR[91] R[100]mm/sec CNT100;
   1:  PR[91,1] = PR[90,1] + 8.546;
   1:  PR[91,2] = PR[90,2] + 6.547;
   1:L PR[91] R[100]mm/sec CNT100;
   1:  PR[91,1] = PR[90,1] + 8.060;
   1:  PR[91,2] = PR[90,2] + 5.505;
   1:L PR[91] R[100]mm/sec CNT100;
   1:  PR[91,1] = PR[90,1] + 7.403;
   1:  PR[91,2] = PR[90,2] + 1.783;
   1:L PR[91] R[100]mm/sec CNT100;
   1:  PR[91,1] = PR[90,1] + 7.037;
   1:  PR[91,2] = PR[90,2] + 0.416;
   1:L PR[91] R[100]mm/sec CNT100;
   1:  PR[91,1] = PR[90,1] + 6.945;
   1:  PR[91,2] = PR[90,2] + -0.641;
   1:L PR[91] R[100]mm/sec CNT100;
   1:  PR[91,1] = PR[90,1] + 7.602;
   1:  PR[91,2] = PR[90,2] + -4.364;
   1:L PR[91] R[100]mm/sec CNT100;
   1:  PR[91,1] = PR[90,1] + 7.725;
   1:  PR[91,2] = PR[90,2] + -5.771;
   1:L PR[91] R[100]mm/sec CNT100;
   1:  PR[91,1] = PR[90,1] + 8.000;
   1:  PR[91,2] = PR[90,2] + -6.800;
   1:L PR[91] R[100]mm/sec CNT100;
   1:  PR[91,1] = PR[90,1] + 9.889;
   1:  PR[91,2] = PR[90,2] + -10.071;
   1:L PR[91] R[100]mm/sec CNT100;
   1:  PR[91,1] = PR[90,1] + 10.487;
   1:  PR[91,2] = PR[90,2] + -11.352;
   1:L PR[91] R[100]mm/sec CNT100;
   1:  PR[91,1] = PR[90,1] + 11.099;
   1:  PR[91,2] = PR[90,2] + -12.225;
   1:L PR[91] R[100]mm/sec CNT100;
   1:  PR[91,1] = PR[90,1] + 13.992;
   1:  PR[91,2] = PR[90,2] + -14.653;
   1:L PR[91] R[100]mm/sec CNT100;
   1:  PR[91,1] = PR[90,1] + 14.990;
   1:  PR[91,2] = PR[90,2] + -15.651;
   1:L PR[91] R[100]mm/sec CNT100;
   1:  PR[91,1] = PR[90,1] + 15.863;
   1:  PR[91,2] = PR[90,2] + -16.262;
   1:L PR[91] R[100]mm/sec CNT100;
   1:  PR[91,1] = PR[90,1] + 19.414;
   1:  PR[91,2] = PR[90,2] + -17.555;
   1:L PR[91] R[100]mm/sec CNT100;
   1:  PR[91,1] = PR[90,1] + 20.693;
   1:  PR[91,2] = PR[90,2] + -18.151;
   1:L PR[91] R[100]mm/sec CNT100;
   1:  PR[91,1] = PR[90,1] + 21.722;
   1:  PR[91,2] = PR[90,2] + -18.426;
   1:L PR[91] R[100]mm/sec CNT100;
   1:  PR[91,1] = PR[90,1] + 25.503;
   1:L PR[91] R[100]mm/sec CNT100;
   1:  PR[91,1] = PR[90,1] + 26.910;
   1:  PR[91,2] = PR[90,2] + -18.549;
   1:L PR[91] R[100]mm/sec CNT100;
   1:  PR[91,1] = PR[90,1] + 27.969;
   1:  PR[91,2] = PR[90,2] + -18.456;
   1:L PR[91] R[100]mm/sec CNT100;
   1:  PR[91,1] = PR[90,1] + 31.519;
   1:  PR[91,2] = PR[90,2] + -17.163;
   1:L PR[91] R[100]mm/sec CNT100;
   1:  PR[91,1] = PR[90,1] + 32.885;
   1:  PR[91,2] = PR[90,2] + -16.796;
   1:L PR[91] R[100]mm/sec CNT100;
   1:  PR[91,1] = PR[90,1] + 33.926;
   1:  PR[91,2] = PR[90,2] + -16.311;
   1:L PR[91] R[100]mm/sec CNT100;
   1:  PR[91,1] = PR[90,1] + 34.942;
   1:  PR[91,2] = PR[90,2] + -15.599;
   1:L PR[91] R[100]mm/sec CNT100;
   1:  PR[91,1] = PR[90,1] + 37.837;
   1:  PR[91,2] = PR[90,2] + -13.170;
   1:L PR[91] R[100]mm/sec CNT100;
   1:  PR[91,1] = PR[90,1] + 38.711;
   1:  PR[91,2] = PR[90,2] + -12.296;
   1:L PR[91] R[100]mm/sec CNT100;
   1:  PR[91,1] = PR[90,1] + 39.423;
   1:  PR[91,2] = PR[90,2] + -11.278;
   1:L PR[91] R[100]mm/sec CNT100;
   1:  PR[91,1] = PR[90,1] + 41.313;
   1:  PR[91,2] = PR[90,2] + -8.006;
   1:L PR[91] R[100]mm/sec CNT100;
   1:  PR[91,1] = PR[90,1] + 41.799;
   1:  PR[91,2] = PR[90,2] + -6.964;
   1:L PR[91] R[100]mm/sec CNT100;
   1:  PR[91,1] = PR[90,1] + 42.456;
   1:  PR[91,2] = PR[90,2] + -3.242;
   1:L PR[91] R[100]mm/sec CNT100;
   1:  PR[91,1] = PR[90,1] + 42.822;
   1:  PR[91,2] = PR[90,2] + -1.875;
   1:L PR[91] R[100]mm/sec CNT100;
   1:  PR[91,1] = PR[90,1] + 42.914;
   1:  PR[91,2] = PR[90,2] + -0.818;
   1:L PR[91] R[100]mm/sec CNT100;
   1:  PR[91,1] = PR[90,1] + 42.257;
   1:  PR[91,2] = PR[90,2] + 2.905;
   1:L PR[91] R[100]mm/sec CNT100;
   1:  PR[91,1] = PR[90,1] + 42.134;
   1:  PR[91,2] = PR[90,2] + 4.312;
   1:L PR[91] R[100]mm/sec CNT100;
   1:  PR[91,1] = PR[90,1] + 41.859;
   1:  PR[91,2] = PR[90,2] + 5.341;
   1:L PR[91] R[100]mm/sec CNT100;
   1:  PR[91,1] = PR[90,1] + 39.969;
   1:  PR[91,2] = PR[90,2] + 8.612;
   1:L PR[91] R[100]mm/sec CNT100;
   1:  PR[91,1] = PR[90,1] + 39.372;
   1:  PR[91,2] = PR[90,2] + 9.893;
   1:L PR[91] R[100]mm/sec CNT100;
   1:  PR[91,1] = PR[90,1] + 38.760;
   1:  PR[91,2] = PR[90,2] + 10.766;
   1:L PR[91] R[100]mm/sec CNT100;
   1:  PR[91,1] = PR[90,1] + 35.867;
   1:  PR[91,2] = PR[90,2] + 13.194;
   1:L PR[91] R[100]mm/sec CNT100;
   1:  PR[91,1] = PR[90,1] + 34.869;
   1:  PR[91,2] = PR[90,2] + 14.192;
   1:L PR[91] R[100]mm/sec CNT100;
   1:  PR[91,1] = PR[90,1] + 33.995;
   1:  PR[91,2] = PR[90,2] + 14.803;
   1:L PR[91] R[100]mm/sec CNT100;
   1:  PR[91,1] = PR[90,1] + 30.445;
   1:  PR[91,2] = PR[90,2] + 16.096;
   1:L PR[91] R[100]mm/sec CNT100;
   1:  PR[91,1] = PR[90,1] + 29.165;
   1:  PR[91,2] = PR[90,2] + 16.692;
   1:L PR[91] R[100]mm/sec CNT100;
   1:  PR[91,1] = PR[90,1] + 28.137;
   1:  PR[91,2] = PR[90,2] + 16.967;
   1:L PR[91] R[100]mm/sec CNT100TB   .50sec,CALL END_PUD;
   1:  PR[92] = PR[91];
   1:  PR[92,3] = PR[92,3] + 20;
   1:J PR[92] 10% FINE;
   1:  PR[91,1] = PR[90,1] + 61.097;
   1:  PR[91,2] = PR[90,2] + -12.223;
   1:  PR[92] = PR[91];
   1:  PR[92,3] = PR[92,3] + 20;
   1:J PR[92] 10% FINE;
   1:L PR[91] R[100]mm/sec CNT100;
   1:  CALL LASER_DRAHT_START;
   1:  PR[91,1] = PR[90,1] + 63.991;
   1:  PR[91,2] = PR[90,2] + -14.652;
   1:L PR[91] R[100]mm/sec CNT100;
   1:  PR[91,1] = PR[90,1] + 64.988;
   1:  PR[91,2] = PR[90,2] + -15.649;
   1:L PR[91] R[100]mm/sec CNT100;
   1:  PR[91,1] = PR[90,1] + 65.860;
   1:  PR[91,2] = PR[90,2] + -16.260;
   1:L PR[91] R[100]mm/sec CNT100;
   1:  PR[91,1] = PR[90,1] + 69.411;
   1:  PR[91,2] = PR[90,2] + -17.553;
   1:L PR[91] R[100]mm/sec CNT100;
   1:  PR[91,1] = PR[90,1] + 70.690;
   1:  PR[91,2] = PR[90,2] + -18.149;
   1:L PR[91] R[100]mm/sec CNT100;
   1:  PR[91,1] = PR[90,1] + 71.802;
   1:  PR[91,2] = PR[90,2] + -18.448;
   1:L PR[91] R[100]mm/sec CNT100;
   1:  PR[91,1] = PR[90,1] + 73.035;
   1:  PR[91,2] = PR[90,2] + -18.556;
   1:L PR[91] R[100]mm/sec CNT100;
   1:  PR[91,1] = PR[90,1] + 76.818;
   1:L PR[91] R[100]mm/sec CNT100;
   1:  PR[91,1] = PR[90,1] + 78.052;
   1:  PR[91,2] = PR[90,2] + -18.449;
   1:L PR[91] R[100]mm/sec CNT100;
   1:  PR[91,1] = PR[90,1] + 79.249;
   1:  PR[91,2] = PR[90,2] + -18.128;
   1:L PR[91] R[100]mm/sec CNT100;
   1:  PR[91,1] = PR[90,1] + 82.801;
   1:  PR[91,2] = PR[90,2] + -16.835;
   1:L PR[91] R[100]mm/sec CNT100;
   1:  PR[91,1] = PR[90,1] + 83.923;
   1:  PR[91,2] = PR[90,2] + -16.312;
   1:L PR[91] R[100]mm/sec CNT100;
   1:  PR[91,1] = PR[90,1] + 84.940;
   1:  PR[91,2] = PR[90,2] + -15.601;
   1:L PR[91] R[100]mm/sec CNT100;
   1:  PR[91,1] = PR[90,1] + 87.834;
   1:  PR[91,2] = PR[90,2] + -13.172;
   1:L PR[91] R[100]mm/sec CNT100;
   1:  PR[91,1] = PR[90,1] + 88.710;
   1:  PR[91,2] = PR[90,2] + -12.297;
   1:L PR[91] R[100]mm/sec CNT100;
   1:  PR[91,1] = PR[90,1] + 89.422;
   1:  PR[91,2] = PR[90,2] + -11.280;
   1:L PR[91] R[100]mm/sec CNT100;
   1:  PR[91,1] = PR[90,1] + 91.312;
   1:  PR[91,2] = PR[90,2] + -8.007;
   1:L PR[91] R[100]mm/sec CNT100;
   1:  PR[91,1] = PR[90,1] + 91.836;
   1:  PR[91,2] = PR[90,2] + -6.885;
   1:L PR[91] R[100]mm/sec CNT100;
   1:  PR[91,1] = PR[90,1] + 92.157;
   1:  PR[91,2] = PR[90,2] + -5.686;
   1:L PR[91] R[100]mm/sec CNT100;
   1:  PR[91,1] = PR[90,1] + 92.814;
   1:  PR[91,2] = PR[90,2] + -1.962;
   1:L PR[91] R[100]mm/sec CNT100;
   1:  PR[91,1] = PR[90,1] + 92.914;
   1:  PR[91,2] = PR[90,2] + -0.818;
   1:L PR[91] R[100]mm/sec CNT100;
   1:  PR[91,1] = PR[90,1] + 92.257;
   1:  PR[91,2] = PR[90,2] + 2.905;
   1:L PR[91] R[100]mm/sec CNT100;
   1:  PR[91,1] = PR[90,1] + 92.134;
   1:  PR[91,2] = PR[90,2] + 4.312;
   1:L PR[91] R[100]mm/sec CNT100;
   1:  PR[91,1] = PR[90,1] + 91.836;
   1:  PR[91,2] = PR[90,2] + 5.426;
   1:L PR[91] R[100]mm/sec CNT100;
   1:  PR[91,1] = PR[90,1] + 91.313;
   1:  PR[91,2] = PR[90,2] + 6.547;
   1:L PR[91] R[100]mm/sec CNT100;
   1:  PR[91,1] = PR[90,1] + 89.423;
   1:  PR[91,2] = PR[90,2] + 9.820;
   1:L PR[91] R[100]mm/sec CNT100;
   1:  PR[91,1] = PR[90,1] + 88.762;
   1:  PR[91,2] = PR[90,2] + 10.765;
   1:L PR[91] R[100]mm/sec CNT100;
   1:  PR[91,1] = PR[90,1] + 85.868;
   1:  PR[91,2] = PR[90,2] + 13.193;
   1:L PR[91] R[100]mm/sec CNT100;
   1:  PR[91,1] = PR[90,1] + 84.870;
   1:  PR[91,2] = PR[90,2] + 14.190;
   1:L PR[91] R[100]mm/sec CNT100;
   1:  PR[91,1] = PR[90,1] + 83.998;
   1:  PR[91,2] = PR[90,2] + 14.801;
   1:L PR[91] R[100]mm/sec CNT100;
   1:  PR[91,1] = PR[90,1] + 80.448;
   1:  PR[91,2] = PR[90,2] + 16.094;
   1:L PR[91] R[100]mm/sec CNT100;
   1:  PR[91,1] = PR[90,1] + 79.169;
   1:  PR[91,2] = PR[90,2] + 16.691;
   1:L PR[91] R[100]mm/sec CNT100;
   1:  PR[91,1] = PR[90,1] + 78.056;
   1:  PR[91,2] = PR[90,2] + 16.989;
   1:L PR[91] R[100]mm/sec CNT100;
   1:  PR[91,1] = PR[90,1] + 76.824;
   1:  PR[91,2] = PR[90,2] + 17.097;
   1:L PR[91] R[100]mm/sec CNT100;
   1:  PR[91,1] = PR[90,1] + 73.041;
   1:L PR[91] R[100]mm/sec CNT100;
   1:  PR[91,1] = PR[90,1] + 71.807;
   1:  PR[91,2] = PR[90,2] + 16.990;
   1:L PR[91] R[100]mm/sec CNT100;
   1:  PR[91,1] = PR[90,1] + 70.609;
   1:  PR[91,2] = PR[90,2] + 16.669;
   1:L PR[91] R[100]mm/sec CNT100;
   1:  PR[91,1] = PR[90,1] + 67.057;
   1:  PR[91,2] = PR[90,2] + 15.376;
   1:L PR[91] R[100]mm/sec CNT100;
   1:  PR[91,1] = PR[90,1] + 65.935;
   1:  PR[91,2] = PR[90,2] + 14.853;
   1:L PR[91] R[100]mm/sec CNT100;
   1:  PR[91,1] = PR[90,1] + 64.919;
   1:  PR[91,2] = PR[90,2] + 14.142;
   1:L PR[91] R[100]mm/sec CNT100;
   1:  PR[91,1] = PR[90,1] + 62.024;
   1:  PR[91,2] = PR[90,2] + 11.713;
   1:L PR[91] R[100]mm/sec CNT100;
   1:  PR[91,1] = PR[90,1] + 61.149;
   1:  PR[91,2] = PR[90,2] + 10.838;
   1:L PR[91] R[100]mm/sec CNT100;
   1:  PR[91,1] = PR[90,1] + 60.436;
   1:  PR[91,2] = PR[90,2] + 9.821;
   1:L PR[91] R[100]mm/sec CNT100;
   1:  PR[91,1] = PR[90,1] + 58.546;
   1:  PR[91,2] = PR[90,2] + 6.549;
   1:L PR[91] R[100]mm/sec CNT100;
   1:  PR[91,1] = PR[90,1] + 58.023;
   1:  PR[91,2] = PR[90,2] + 5.426;
   1:L PR[91] R[100]mm/sec CNT100;
   1:  PR[91,1] = PR[90,1] + 57.702;
   1:  PR[91,2] = PR[90,2] + 4.227;
   1:L PR[91] R[100]mm/sec CNT100;
   1:  PR[91,1] = PR[90,1] + 57.045;
   1:  PR[91,2] = PR[90,2] + 0.503;
   1:L PR[91] R[100]mm/sec CNT100;
   1:  PR[91,1] = PR[90,1] + 56.945;
   1:  PR[91,2] = PR[90,2] + -0.641;
   1:L PR[91] R[100]mm/sec CNT100;
   1:  PR[91,1] = PR[90,1] + 57.602;
   1:  PR[91,2] = PR[90,2] + -4.364;
   1:L PR[91] R[100]mm/sec CNT100;
   1:  PR[91,1] = PR[90,1] + 57.724;
   1:  PR[91,2] = PR[90,2] + -5.771;
   1:L PR[91] R[100]mm/sec CNT100;
   1:  PR[91,1] = PR[90,1] + 58.023;
   1:  PR[91,2] = PR[90,2] + -6.884;
   1:L PR[91] R[100]mm/sec CNT100;
   1:  PR[91,1] = PR[90,1] + 58.546;
   1:  PR[91,2] = PR[90,2] + -8.006;
   1:L PR[91] R[100]mm/sec CNT100;
   1:  PR[91,1] = PR[90,1] + 60.436;
   1:  PR[91,2] = PR[90,2] + -11.278;
   1:L PR[91] R[100]mm/sec CNT100;
   1:  PR[91,1] = PR[90,1] + 61.097;
   1:  PR[91,2] = PR[90,2] + -12.223;
   1:L PR[91] R[100]mm/sec CNT100TB   .50sec,CALL END_PUD;
   1:  PR[92] = PR[91];
   1:  PR[92,3] = PR[92,3] + 20;
   1:J PR[92] 10% FINE;
   1:  PR[91] = PR[90];
   1:  PR[91,1] = PR[90,1] + -59.466;
   1:  PR[91,2] = PR[90,2] + 7.635;
   1:  PR[91,3] = PR[90,3] + 5.395;
   1:  PR[92] = PR[91];
   1:  PR[92,3] = PR[92,3] + 20;
   1:J PR[92] 10% FINE;
   1:L PR[91] R[100]mm/sec CNT100;
   1:  CALL LASER_DRAHT_START;
   1:  PR[91,1] = PR[90,1] + -60.303;
   1:  PR[91,2] = PR[90,2] + 9.429;
   1:L PR[91] R[100]mm/sec CNT100;
   1:  PR[91,1] = PR[90,1] + -61.240;
   1:  PR[91,2] = PR[90,2] + 10.767;
   1:L PR[91] R[100]mm/sec CNT100;
   1:  PR[91,1] = PR[90,1] + -63.270;
   1:  PR[91,2] = PR[90,2] + 12.470;
   1:L PR[91] R[100]mm/sec CNT100;
   1:  PR[91,1] = PR[90,1] + -64.668;
   1:  PR[91,2] = PR[90,2] + 13.868;
   1:L PR[91] R[100]mm/sec CNT100;
   1:  PR[91,1] = PR[90,1] + -66.006;
   1:  PR[91,2] = PR[90,2] + 14.804;
   1:L PR[91] R[100]mm/sec CNT100;
   1:  PR[91,1] = PR[90,1] + -68.496;
   1:  PR[91,2] = PR[90,2] + 15.711;
   1:L PR[91] R[100]mm/sec CNT100;
   1:  PR[91,1] = PR[90,1] + -70.289;
   1:  PR[91,2] = PR[90,2] + 16.546;
   1:L PR[91] R[100]mm/sec CNT100;
   1:  PR[91,1] = PR[90,1] + -71.865;
   1:  PR[91,2] = PR[90,2] + 16.967;
   1:L PR[91] R[100]mm/sec CNT100;
   1:  PR[91,1] = PR[90,1] + -74.516;
   1:L PR[91] R[100]mm/sec CNT100;
   1:  PR[91,1] = PR[90,1] + -76.488;
   1:  PR[91,2] = PR[90,2] + 17.139;
   1:L PR[91] R[100]mm/sec CNT100;
   1:  PR[91,1] = PR[90,1] + -78.110;
   1:  PR[91,2] = PR[90,2] + 16.997;
   1:L PR[91] R[100]mm/sec CNT100;
   1:  PR[91,1] = PR[90,1] + -80.600;
   1:  PR[91,2] = PR[90,2] + 16.090;
   1:L PR[91] R[100]mm/sec CNT100;
   1:  PR[91,1] = PR[90,1] + -82.513;
   1:  PR[91,2] = PR[90,2] + 15.577;
   1:L PR[91] R[100]mm/sec CNT100;
   1:  PR[91,1] = PR[90,1] + -84.067;
   1:  PR[91,2] = PR[90,2] + 14.852;
   1:L PR[91] R[100]mm/sec CNT100;
   1:  PR[91,1] = PR[90,1] + -85.548;
   1:  PR[91,2] = PR[90,2] + 13.815;
   1:L PR[91] R[100]mm/sec CNT100;
   1:  PR[91,1] = PR[90,1] + -87.578;
   1:  PR[91,2] = PR[90,2] + 12.111;
   1:L PR[91] R[100]mm/sec CNT100;
   1:  PR[91,1] = PR[90,1] + -88.852;
   1:  PR[91,2] = PR[90,2] + 10.837;
   1:L PR[91] R[100]mm/sec CNT100;
   1:  PR[91,1] = PR[90,1] + -89.890;
   1:  PR[91,2] = PR[90,2] + 9.355;
   1:L PR[91] R[100]mm/sec CNT100;
   1:  PR[91,1] = PR[90,1] + -91.215;
   1:  PR[91,2] = PR[90,2] + 7.060;
   1:L PR[91] R[100]mm/sec CNT100;
   1:  PR[91,1] = PR[90,1] + -91.940;
   1:  PR[91,2] = PR[90,2] + 5.505;
   1:L PR[91] R[100]mm/sec CNT100;
   1:  PR[91,1] = PR[90,1] + -92.401;
   1:  PR[91,2] = PR[90,2] + 2.894;
   1:L PR[91] R[100]mm/sec CNT100;
   1:  PR[91,1] = PR[90,1] + -92.914;
   1:  PR[91,2] = PR[90,2] + 0.979;
   1:L PR[91] R[100]mm/sec CNT100;
   1:  PR[91,1] = PR[90,1] + -93.055;
   1:  PR[91,2] = PR[90,2] + -0.641;
   1:L PR[91] R[100]mm/sec CNT100;
   1:  PR[91,1] = PR[90,1] + -92.595;
   1:  PR[91,2] = PR[90,2] + -3.252;
   1:L PR[91] R[100]mm/sec CNT100;
   1:  PR[91,1] = PR[90,1] + -92.422;
   1:  PR[91,2] = PR[90,2] + -5.222;
   1:L PR[91] R[100]mm/sec CNT100;
   1:  PR[91,1] = PR[90,1] + -92.000;
   1:  PR[91,2] = PR[90,2] + -6.800;
   1:L PR[91] R[100]mm/sec CNT100;
   1:  PR[91,1] = PR[90,1] + -90.675;
   1:  PR[91,2] = PR[90,2] + -9.094;
   1:L PR[91] R[100]mm/sec CNT100;
   1:  PR[91,1] = PR[90,1] + -89.838;
   1:  PR[91,2] = PR[90,2] + -10.888;
   1:L PR[91] R[100]mm/sec CNT100;
   1:  PR[91,1] = PR[90,1] + -88.901;
   1:  PR[91,2] = PR[90,2] + -12.226;
   1:L PR[91] R[100]mm/sec CNT100;
   1:  PR[91,1] = PR[90,1] + -86.872;
   1:  PR[91,2] = PR[90,2] + -13.929;
   1:L PR[91] R[100]mm/sec CNT100;
   1:  PR[91,1] = PR[90,1] + -85.473;
   1:  PR[91,2] = PR[90,2] + -15.327;
   1:L PR[91] R[100]mm/sec CNT100;
   1:  PR[91,1] = PR[90,1] + -84.135;
   1:  PR[91,2] = PR[90,2] + -16.263;
   1:L PR[91] R[100]mm/sec CNT100;
   1:  PR[91,1] = PR[90,1] + -81.645;
   1:  PR[91,2] = PR[90,2] + -17.170;
   1:L PR[91] R[100]mm/sec CNT100;
   1:  PR[91,1] = PR[90,1] + -79.853;
   1:  PR[91,2] = PR[90,2] + -18.005;
   1:L PR[91] R[100]mm/sec CNT100;
   1:  PR[91,1] = PR[90,1] + -78.276;
   1:  PR[91,2] = PR[90,2] + -18.426;
   1:L PR[91] R[100]mm/sec CNT100;
   1:  PR[91,1] = PR[90,1] + -75.625;
   1:L PR[91] R[100]mm/sec CNT100;
   1:  PR[91,1] = PR[90,1] + -73.653;
   1:  PR[91,2] = PR[90,2] + -18.598;
   1:L PR[91] R[100]mm/sec CNT100;
   1:  PR[91,1] = PR[90,1] + -72.031;
   1:  PR[91,2] = PR[90,2] + -18.456;
   1:L PR[91] R[100]mm/sec CNT100;
   1:  PR[91,1] = PR[90,1] + -69.541;
   1:  PR[91,2] = PR[90,2] + -17.549;
   1:L PR[91] R[100]mm/sec CNT100;
   1:  PR[91,1] = PR[90,1] + -67.628;
   1:  PR[91,2] = PR[90,2] + -17.036;
   1:L PR[91] R[100]mm/sec CNT100;
   1:  PR[91,1] = PR[90,1] + -66.074;
   1:  PR[91,2] = PR[90,2] + -16.311;
   1:L PR[91] R[100]mm/sec CNT100;
   1:  PR[91,1] = PR[90,1] + -64.594;
   1:  PR[91,2] = PR[90,2] + -15.274;
   1:L PR[91] R[100]mm/sec CNT100;
   1:  PR[91,1] = PR[90,1] + -62.563;
   1:  PR[91,2] = PR[90,2] + -13.570;
   1:L PR[91] R[100]mm/sec CNT100;
   1:  PR[91,1] = PR[90,1] + -61.289;
   1:  PR[91,2] = PR[90,2] + -12.296;
   1:L PR[91] R[100]mm/sec CNT100;
   1:  PR[91,1] = PR[90,1] + -60.251;
   1:  PR[91,2] = PR[90,2] + -10.814;
   1:L PR[91] R[100]mm/sec CNT100;
   1:  PR[91,1] = PR[90,1] + -58.926;
   1:  PR[91,2] = PR[90,2] + -8.519;
   1:L PR[91] R[100]mm/sec CNT100;
   1:  PR[91,1] = PR[90,1] + -58.201;
   1:  PR[91,2] = PR[90,2] + -6.964;
   1:L PR[91] R[100]mm/sec CNT100;
   1:  PR[91,1] = PR[90,1] + -57.740;
   1:  PR[91,2] = PR[90,2] + -4.353;
   1:L PR[91] R[100]mm/sec CNT100;
   1:  PR[91,1] = PR[90,1] + -57.227;
   1:  PR[91,2] = PR[90,2] + -2.438;
   1:L PR[91] R[100]mm/sec CNT100;
   1:  PR[91,1] = PR[90,1] + -57.086;
   1:  PR[91,2] = PR[90,2] + -0.818;
   1:L PR[91] R[100]mm/sec CNT100;
   1:  PR[91,1] = PR[90,1] + -57.547;
   1:  PR[91,2] = PR[90,2] + 1.793;
   1:L PR[91] R[100]mm/sec CNT100;
   1:  PR[91,1] = PR[90,1] + -57.719;
   1:  PR[91,2] = PR[90,2] + 3.764;
   1:L PR[91] R[100]mm/sec CNT100;
   1:  PR[91,1] = PR[90,1] + -58.141;
   1:  PR[91,2] = PR[90,2] + 5.341;
   1:L PR[91] R[100]mm/sec CNT100;
   1:  PR[91,1] = PR[90,1] + -59.466;
   1:  PR[91,2] = PR[90,2] + 7.635;
   1:L PR[91] R[100]mm/sec CNT100TB   .50sec,CALL END_PUD;
   1:  PR[92] = PR[91];
   1:  PR[92,3] = PR[92,3] + 20;
   1:J PR[92] 10% FINE;
   1:  PR[91,1] = PR[90,1] + -37.639;
   1:  PR[91,2] = PR[90,2] + 12.050;
   1:  PR[92] = PR[91];
   1:  PR[92,3] = PR[92,3] + 20;
   1:J PR[92] 10% FINE;
   1:L PR[91] R[100]mm/sec CNT100;
   1:  CALL LASER_DRAHT_START;
   1:  PR[91,1] = PR[90,1] + -38.792;
   1:  PR[91,2] = PR[90,2] + 10.897;
   1:L PR[91] R[100]mm/sec CNT100;
   1:  PR[91,1] = PR[90,1] + -40.117;
   1:  PR[91,2] = PR[90,2] + 8.602;
   1:L PR[91] R[100]mm/sec CNT100;
   1:  PR[91,1] = PR[90,1] + -41.252;
   1:  PR[91,2] = PR[90,2] + 6.981;
   1:L PR[91] R[100]mm/sec CNT100;
   1:  PR[91,1] = PR[90,1] + -41.941;
   1:  PR[91,2] = PR[90,2] + 5.503;
   1:L PR[91] R[100]mm/sec CNT100;
   1:  PR[91,1] = PR[90,1] + -42.402;
   1:  PR[91,2] = PR[90,2] + 2.892;
   1:L PR[91] R[100]mm/sec CNT100;
   1:  PR[91,1] = PR[90,1] + -42.914;
   1:  PR[91,2] = PR[90,2] + 0.980;
   1:L PR[91] R[100]mm/sec CNT100;
   1:  PR[91,1] = PR[90,1] + -43.055;
   1:  PR[91,2] = PR[90,2] + -0.641;
   1:L PR[91] R[100]mm/sec CNT100;
   1:  PR[91,1] = PR[90,1] + -42.595;
   1:  PR[91,2] = PR[90,2] + -3.252;
   1:L PR[91] R[100]mm/sec CNT100;
   1:  PR[91,1] = PR[90,1] + -42.422;
   1:  PR[91,2] = PR[90,2] + -5.222;
   1:L PR[91] R[100]mm/sec CNT100;
   1:  PR[91,1] = PR[90,1] + -41.978;
   1:  PR[91,2] = PR[90,2] + -6.882;
   1:L PR[91] R[100]mm/sec CNT100;
   1:  PR[91,1] = PR[90,1] + -41.215;
   1:  PR[91,2] = PR[90,2] + -8.519;
   1:L PR[91] R[100]mm/sec CNT100;
   1:  PR[91,1] = PR[90,1] + -39.890;
   1:  PR[91,2] = PR[90,2] + -10.814;
   1:L PR[91] R[100]mm/sec CNT100;
   1:  PR[91,1] = PR[90,1] + -38.855;
   1:  PR[91,2] = PR[90,2] + -12.293;
   1:L PR[91] R[100]mm/sec CNT100;
   1:  PR[91,1] = PR[90,1] + -37.578;
   1:  PR[91,2] = PR[90,2] + -13.570;
   1:L PR[91] R[100]mm/sec CNT100;
   1:  PR[91,1] = PR[90,1] + -35.547;
   1:  PR[91,2] = PR[90,2] + -15.274;
   1:L PR[91] R[100]mm/sec CNT100;
   1:  PR[91,1] = PR[90,1] + -34.070;
   1:  PR[91,2] = PR[90,2] + -16.309;
   1:L PR[91] R[100]mm/sec CNT100;
   1:  PR[91,1] = PR[90,1] + -32.433;
   1:  PR[91,2] = PR[90,2] + -17.073;
   1:L PR[91] R[100]mm/sec CNT100;
   1:  PR[91,1] = PR[90,1] + -29.941;
   1:  PR[91,2] = PR[90,2] + -17.980;
   1:L PR[91] R[100]mm/sec CNT100;
   1:  PR[91,1] = PR[90,1] + -28.197;
   1:  PR[91,2] = PR[90,2] + -18.448;
   1:L PR[91] R[100]mm/sec CNT100;
   1:  PR[91,1] = PR[90,1] + -26.397;
   1:  PR[91,2] = PR[90,2] + -18.606;
   1:L PR[91] R[100]mm/sec CNT100;
   1:  PR[91,1] = PR[90,1] + -23.745;
   1:L PR[91] R[100]mm/sec CNT100;
   1:  PR[91,1] = PR[90,1] + -22.033;
   1:  PR[91,2] = PR[90,2] + -18.456;
   1:L PR[91] R[100]mm/sec CNT100;
   1:  PR[91,1] = PR[90,1] + -19.543;
   1:  PR[91,2] = PR[90,2] + -17.549;
   1:L PR[91] R[100]mm/sec CNT100;
   1:  PR[91,1] = PR[90,1] + -17.630;
   1:  PR[91,2] = PR[90,2] + -17.036;
   1:L PR[91] R[100]mm/sec CNT100;
   1:  PR[91,1] = PR[90,1] + -16.152;
   1:  PR[91,2] = PR[90,2] + -16.347;
   1:L PR[91] R[100]mm/sec CNT100;
   1:  PR[91,1] = PR[90,1] + -14.123;
   1:  PR[91,2] = PR[90,2] + -14.644;
   1:L PR[91] R[100]mm/sec CNT100;
   1:  PR[91,1] = PR[90,1] + -12.502;
   1:  PR[91,2] = PR[90,2] + -13.509;
   1:L PR[91] R[100]mm/sec CNT100;
   1:  PR[91,1] = PR[90,1] + -11.349;
   1:  PR[91,2] = PR[90,2] + -12.356;
   1:L PR[91] R[100]mm/sec CNT100;
   1:  PR[91,1] = PR[90,1] + -10.024;
   1:  PR[91,2] = PR[90,2] + -10.061;
   1:L PR[91] R[100]mm/sec CNT100;
   1:  PR[91,1] = PR[90,1] + -8.889;
   1:  PR[91,2] = PR[90,2] + -8.440;
   1:L PR[91] R[100]mm/sec CNT100;
   1:  PR[91,1] = PR[90,1] + -8.200;
   1:  PR[91,2] = PR[90,2] + -6.962;
   1:L PR[91] R[100]mm/sec CNT100;
   1:  PR[91,1] = PR[90,1] + -7.740;
   1:  PR[91,2] = PR[90,2] + -4.351;
   1:L PR[91] R[100]mm/sec CNT100;
   1:  PR[91,1] = PR[90,1] + -7.228;
   1:  PR[91,2] = PR[90,2] + -2.439;
   1:L PR[91] R[100]mm/sec CNT100;
   1:  PR[91,1] = PR[90,1] + -7.086;
   1:  PR[91,2] = PR[90,2] + -0.818;
   1:L PR[91] R[100]mm/sec CNT100;
   1:  PR[91,1] = PR[90,1] + -7.547;
   1:  PR[91,2] = PR[90,2] + 1.793;
   1:L PR[91] R[100]mm/sec CNT100;
   1:  PR[91,1] = PR[90,1] + -7.719;
   1:  PR[91,2] = PR[90,2] + 3.764;
   1:L PR[91] R[100]mm/sec CNT100;
   1:  PR[91,1] = PR[90,1] + -8.163;
   1:  PR[91,2] = PR[90,2] + 5.423;
   1:L PR[91] R[100]mm/sec CNT100;
   1:  PR[91,1] = PR[90,1] + -8.926;
   1:  PR[91,2] = PR[90,2] + 7.060;
   1:L PR[91] R[100]mm/sec CNT100;
   1:  PR[91,1] = PR[90,1] + -10.251;
   1:  PR[91,2] = PR[90,2] + 9.355;
   1:L PR[91] R[100]mm/sec CNT100;
   1:  PR[91,1] = PR[90,1] + -11.286;
   1:  PR[91,2] = PR[90,2] + 10.834;
   1:L PR[91] R[100]mm/sec CNT100;
   1:  PR[91,1] = PR[90,1] + -12.563;
   1:  PR[91,2] = PR[90,2] + 12.112;
   1:L PR[91] R[100]mm/sec CNT100;
   1:  PR[91,1] = PR[90,1] + -14.594;
   1:  PR[91,2] = PR[90,2] + 13.815;
   1:L PR[91] R[100]mm/sec CNT100;
   1:  PR[91,1] = PR[90,1] + -16.072;
   1:  PR[91,2] = PR[90,2] + 14.851;
   1:L PR[91] R[100]mm/sec CNT100;
   1:  PR[91,1] = PR[90,1] + -17.709;
   1:  PR[91,2] = PR[90,2] + 15.614;
   1:L PR[91] R[100]mm/sec CNT100;
   1:  PR[91,1] = PR[90,1] + -20.200;
   1:  PR[91,2] = PR[90,2] + 16.522;
   1:L PR[91] R[100]mm/sec CNT100;
   1:  PR[91,1] = PR[90,1] + -21.944;
   1:  PR[91,2] = PR[90,2] + 16.989;
   1:L PR[91] R[100]mm/sec CNT100;
   1:  PR[91,1] = PR[90,1] + -23.744;
   1:  PR[91,2] = PR[90,2] + 17.147;
   1:L PR[91] R[100]mm/sec CNT100;
   1:  PR[91,1] = PR[90,1] + -26.397;
   1:L PR[91] R[100]mm/sec CNT100;
   1:  PR[91,1] = PR[90,1] + -28.109;
   1:  PR[91,2] = PR[90,2] + 16.997;
   1:L PR[91] R[100]mm/sec CNT100;
   1:  PR[91,1] = PR[90,1] + -30.599;
   1:  PR[91,2] = PR[90,2] + 16.090;
   1:L PR[91] R[100]mm/sec CNT100;
   1:  PR[91,1] = PR[90,1] + -32.511;
   1:  PR[91,2] = PR[90,2] + 15.578;
   1:L PR[91] R[100]mm/sec CNT100;
   1:  PR[91,1] = PR[90,1] + -33.989;
   1:  PR[91,2] = PR[90,2] + 14.888;
   1:L PR[91] R[100]mm/sec CNT100;
   1:  PR[91,1] = PR[90,1] + -36.018;
   1:  PR[91,2] = PR[90,2] + 13.185;
   1:L PR[91] R[100]mm/sec CNT100;
   1:  PR[91,1] = PR[90,1] + -37.639;
   1:  PR[91,2] = PR[90,2] + 12.050;
   1:L PR[91] R[100]mm/sec CNT100TB   .50sec,CALL END_PUD;
   1:  PR[92] = PR[91];
   1:  PR[92,3] = PR[92,3] + 20;
   1:J PR[92] 10% FINE;
   1:  PR[91,1] = PR[90,1] + 29.712;
   1:  PR[91,2] = PR[90,2] + 16.546;
   1:  PR[92] = PR[91];
   1:  PR[92,3] = PR[92,3] + 20;
   1:J PR[92] 10% FINE;
   1:L PR[91] R[100]mm/sec CNT100;
   1:  CALL LASER_DRAHT_START;
   1:  PR[91,1] = PR[90,1] + 28.135;
   1:  PR[91,2] = PR[90,2] + 16.967;
   1:L PR[91] R[100]mm/sec CNT100;
   1:  PR[91,1] = PR[90,1] + 25.484;
   1:L PR[91] R[100]mm/sec CNT100;
   1:  PR[91,1] = PR[90,1] + 23.512;
   1:  PR[91,2] = PR[90,2] + 17.139;
   1:L PR[91] R[100]mm/sec CNT100;
   1:  PR[91,1] = PR[90,1] + 21.890;
   1:  PR[91,2] = PR[90,2] + 16.997;
   1:L PR[91] R[100]mm/sec CNT100;
   1:  PR[91,1] = PR[90,1] + 19.400;
   1:  PR[91,2] = PR[90,2] + 16.090;
   1:L PR[91] R[100]mm/sec CNT100;
   1:  PR[91,1] = PR[90,1] + 17.487;
   1:  PR[91,2] = PR[90,2] + 15.577;
   1:L PR[91] R[100]mm/sec CNT100;
   1:  PR[91,1] = PR[90,1] + 15.933;
   1:  PR[91,2] = PR[90,2] + 14.852;
   1:L PR[91] R[100]mm/sec CNT100;
   1:  PR[91,1] = PR[90,1] + 14.452;
   1:  PR[91,2] = PR[90,2] + 13.815;
   1:L PR[91] R[100]mm/sec CNT100;
   1:  PR[91,1] = PR[90,1] + 12.422;
   1:  PR[91,2] = PR[90,2] + 12.111;
   1:L PR[91] R[100]mm/sec CNT100;
   1:  PR[91,1] = PR[90,1] + 11.148;
   1:  PR[91,2] = PR[90,2] + 10.837;
   1:L PR[91] R[100]mm/sec CNT100;
   1:  PR[91,1] = PR[90,1] + 10.110;
   1:  PR[91,2] = PR[90,2] + 9.355;
   1:L PR[91] R[100]mm/sec CNT100;
   1:  PR[91,1] = PR[90,1] + 8.785;
   1:  PR[91,2] = PR[90,2] + 7.060;
   1:L PR[91] R[100]mm/sec CNT100;
   1:  PR[91,1] = PR[90,1] + 8.060;
   1:  PR[91,2] = PR[90,2] + 5.505;
   1:L PR[91] R[100]mm/sec CNT100;
   1:  PR[91,1] = PR[90,1] + 7.599;
   1:  PR[91,2] = PR[90,2] + 2.894;
   1:L PR[91] R[100]mm/sec CNT100;
   1:  PR[91,1] = PR[90,1] + 7.086;
   1:  PR[91,2] = PR[90,2] + 0.979;
   1:L PR[91] R[100]mm/sec CNT100;
   1:  PR[91,1] = PR[90,1] + 6.945;
   1:  PR[91,2] = PR[90,2] + -0.641;
   1:L PR[91] R[100]mm/sec CNT100;
   1:  PR[91,1] = PR[90,1] + 7.405;
   1:  PR[91,2] = PR[90,2] + -3.252;
   1:L PR[91] R[100]mm/sec CNT100;
   1:  PR[91,1] = PR[90,1] + 7.578;
   1:  PR[91,2] = PR[90,2] + -5.222;
   1:L PR[91] R[100]mm/sec CNT100;
   1:  PR[91,1] = PR[90,1] + 8.000;
   1:  PR[91,2] = PR[90,2] + -6.800;
   1:L PR[91] R[100]mm/sec CNT100;
   1:  PR[91,1] = PR[90,1] + 9.325;
   1:  PR[91,2] = PR[90,2] + -9.094;
   1:L PR[91] R[100]mm/sec CNT100;
   1:  PR[91,1] = PR[90,1] + 10.162;
   1:  PR[91,2] = PR[90,2] + -10.888;
   1:L PR[91] R[100]mm/sec CNT100;
   1:  PR[91,1] = PR[90,1] + 11.099;
   1:  PR[91,2] = PR[90,2] + -12.226;
   1:L PR[91] R[100]mm/sec CNT100;
   1:  PR[91,1] = PR[90,1] + 13.128;
   1:  PR[91,2] = PR[90,2] + -13.929;
   1:L PR[91] R[100]mm/sec CNT100;
   1:  PR[91,1] = PR[90,1] + 14.527;
   1:  PR[91,2] = PR[90,2] + -15.327;
   1:L PR[91] R[100]mm/sec CNT100;
   1:  PR[91,1] = PR[90,1] + 15.865;
   1:  PR[91,2] = PR[90,2] + -16.263;
   1:L PR[91] R[100]mm/sec CNT100;
   1:  PR[91,1] = PR[90,1] + 18.355;
   1:  PR[91,2] = PR[90,2] + -17.169;
   1:L PR[91] R[100]mm/sec CNT100;
   1:  PR[91,1] = PR[90,1] + 20.147;
   1:  PR[91,2] = PR[90,2] + -18.004;
   1:L PR[91] R[100]mm/sec CNT100;
   1:  PR[91,1] = PR[90,1] + 21.724;
   1:  PR[91,2] = PR[90,2] + -18.426;
   1:L PR[91] R[100]mm/sec CNT100;
   1:  PR[91,1] = PR[90,1] + 24.375;
   1:L PR[91] R[100]mm/sec CNT100;
   1:  PR[91,1] = PR[90,1] + 26.347;
   1:  PR[91,2] = PR[90,2] + -18.598;
   1:L PR[91] R[100]mm/sec CNT100;
   1:  PR[91,1] = PR[90,1] + 27.969;
   1:  PR[91,2] = PR[90,2] + -18.456;
   1:L PR[91] R[100]mm/sec CNT100;
   1:  PR[91,1] = PR[90,1] + 30.459;
   1:  PR[91,2] = PR[90,2] + -17.549;
   1:L PR[91] R[100]mm/sec CNT100;
   1:  PR[91,1] = PR[90,1] + 32.372;
   1:  PR[91,2] = PR[90,2] + -17.036;
   1:L PR[91] R[100]mm/sec CNT100;
   1:  PR[91,1] = PR[90,1] + 33.926;
   1:  PR[91,2] = PR[90,2] + -16.311;
   1:L PR[91] R[100]mm/sec CNT100;
   1:  PR[91,1] = PR[90,1] + 35.406;
   1:  PR[91,2] = PR[90,2] + -15.274;
   1:L PR[91] R[100]mm/sec CNT100;
   1:  PR[91,1] = PR[90,1] + 37.437;
   1:  PR[91,2] = PR[90,2] + -13.570;
   1:L PR[91] R[100]mm/sec CNT100;
   1:  PR[91,1] = PR[90,1] + 38.711;
   1:  PR[91,2] = PR[90,2] + -12.296;
   1:L PR[91] R[100]mm/sec CNT100;
   1:  PR[91,1] = PR[90,1] + 39.749;
   1:  PR[91,2] = PR[90,2] + -10.814;
   1:L PR[91] R[100]mm/sec CNT100;
   1:  PR[91,1] = PR[90,1] + 41.074;
   1:  PR[91,2] = PR[90,2] + -8.519;
   1:L PR[91] R[100]mm/sec CNT100;
   1:  PR[91,1] = PR[90,1] + 41.799;
   1:  PR[91,2] = PR[90,2] + -6.964;
   1:L PR[91] R[100]mm/sec CNT100;
   1:  PR[91,1] = PR[90,1] + 42.260;
   1:  PR[91,2] = PR[90,2] + -4.353;
   1:L PR[91] R[100]mm/sec CNT100;
   1:  PR[91,1] = PR[90,1] + 42.773;
   1:  PR[91,2] = PR[90,2] + -2.438;
   1:L PR[91] R[100]mm/sec CNT100;
   1:  PR[91,1] = PR[90,1] + 42.914;
   1:  PR[91,2] = PR[90,2] + -0.818;
   1:L PR[91] R[100]mm/sec CNT100;
   1:  PR[91,1] = PR[90,1] + 42.453;
   1:  PR[91,2] = PR[90,2] + 1.793;
   1:L PR[91] R[100]mm/sec CNT100;
   1:  PR[91,1] = PR[90,1] + 42.281;
   1:  PR[91,2] = PR[90,2] + 3.764;
   1:L PR[91] R[100]mm/sec CNT100;
   1:  PR[91,1] = PR[90,1] + 41.859;
   1:  PR[91,2] = PR[90,2] + 5.341;
   1:L PR[91] R[100]mm/sec CNT100;
   1:  PR[91,1] = PR[90,1] + 40.534;
   1:  PR[91,2] = PR[90,2] + 7.635;
   1:L PR[91] R[100]mm/sec CNT100;
   1:  PR[91,1] = PR[90,1] + 39.697;
   1:  PR[91,2] = PR[90,2] + 9.429;
   1:L PR[91] R[100]mm/sec CNT100;
   1:  PR[91,1] = PR[90,1] + 38.760;
   1:  PR[91,2] = PR[90,2] + 10.767;
   1:L PR[91] R[100]mm/sec CNT100;
   1:  PR[91,1] = PR[90,1] + 36.730;
   1:  PR[91,2] = PR[90,2] + 12.470;
   1:L PR[91] R[100]mm/sec CNT100;
   1:  PR[91,1] = PR[90,1] + 35.332;
   1:  PR[91,2] = PR[90,2] + 13.868;
   1:L PR[91] R[100]mm/sec CNT100;
   1:  PR[91,1] = PR[90,1] + 33.994;
   1:  PR[91,2] = PR[90,2] + 14.804;
   1:L PR[91] R[100]mm/sec CNT100;
   1:  PR[91,1] = PR[90,1] + 31.504;
   1:  PR[91,2] = PR[90,2] + 15.711;
   1:L PR[91] R[100]mm/sec CNT100;
   1:  PR[91,1] = PR[90,1] + 29.712;
   1:  PR[91,2] = PR[90,2] + 16.546;
   1:L PR[91] R[100]mm/sec CNT100TB   .50sec,CALL END_PUD;
   1:  PR[92] = PR[91];
   1:  PR[92,3] = PR[92,3] + 20;
   1:J PR[92] 10% FINE;
   1:  PR[91,1] = PR[90,1] + 88.761;
   1:  PR[91,2] = PR[90,2] + 10.765;
   1:  PR[92] = PR[91];
   1:  PR[92,3] = PR[92,3] + 20;
   1:J PR[92] 10% FINE;
   1:L PR[91] R[100]mm/sec CNT100;
   1:  CALL LASER_DRAHT_START;
   1:  PR[91,1] = PR[90,1] + 86.732;
   1:  PR[91,2] = PR[90,2] + 12.468;
   1:L PR[91] R[100]mm/sec CNT100;
   1:  PR[91,1] = PR[90,1] + 85.335;
   1:  PR[91,2] = PR[90,2] + 13.865;
   1:L PR[91] R[100]mm/sec CNT100;
   1:  PR[91,1] = PR[90,1] + 83.998;
   1:  PR[91,2] = PR[90,2] + 14.801;
   1:L PR[91] R[100]mm/sec CNT100;
   1:  PR[91,1] = PR[90,1] + 81.508;
   1:  PR[91,2] = PR[90,2] + 15.708;
   1:L PR[91] R[100]mm/sec CNT100;
   1:  PR[91,1] = PR[90,1] + 79.717;
   1:  PR[91,2] = PR[90,2] + 16.544;
   1:L PR[91] R[100]mm/sec CNT100;
   1:  PR[91,1] = PR[90,1] + 78.057;
   1:  PR[91,2] = PR[90,2] + 16.989;
   1:L PR[91] R[100]mm/sec CNT100;
   1:  PR[91,1] = PR[90,1] + 76.260;
   1:  PR[91,2] = PR[90,2] + 17.147;
   1:L PR[91] R[100]mm/sec CNT100;
   1:  PR[91,1] = PR[90,1] + 73.607;
   1:L PR[91] R[100]mm/sec CNT100;
   1:  PR[91,1] = PR[90,1] + 71.809;
   1:  PR[91,2] = PR[90,2] + 16.990;
   1:L PR[91] R[100]mm/sec CNT100;
   1:  PR[91,1] = PR[90,1] + 70.063;
   1:  PR[91,2] = PR[90,2] + 16.523;
   1:L PR[91] R[100]mm/sec CNT100;
   1:  PR[91,1] = PR[90,1] + 67.572;
   1:  PR[91,2] = PR[90,2] + 15.616;
   1:L PR[91] R[100]mm/sec CNT100;
   1:  PR[91,1] = PR[90,1] + 65.937;
   1:  PR[91,2] = PR[90,2] + 14.854;
   1:L PR[91] R[100]mm/sec CNT100;
   1:  PR[91,1] = PR[90,1] + 64.455;
   1:  PR[91,2] = PR[90,2] + 13.818;
   1:L PR[91] R[100]mm/sec CNT100;
   1:  PR[91,1] = PR[90,1] + 62.425;
   1:  PR[91,2] = PR[90,2] + 12.114;
   1:L PR[91] R[100]mm/sec CNT100;
   1:  PR[91,1] = PR[90,1] + 61.150;
   1:  PR[91,2] = PR[90,2] + 10.839;
   1:L PR[91] R[100]mm/sec CNT100;
   1:  PR[91,1] = PR[90,1] + 60.111;
   1:  PR[91,2] = PR[90,2] + 9.357;
   1:L PR[91] R[100]mm/sec CNT100;
   1:  PR[91,1] = PR[90,1] + 58.786;
   1:  PR[91,2] = PR[90,2] + 7.062;
   1:L PR[91] R[100]mm/sec CNT100;
   1:  PR[91,1] = PR[90,1] + 58.023;
   1:  PR[91,2] = PR[90,2] + 5.426;
   1:L PR[91] R[100]mm/sec CNT100;
   1:  PR[91,1] = PR[90,1] + 57.555;
   1:  PR[91,2] = PR[90,2] + 3.679;
   1:L PR[91] R[100]mm/sec CNT100;
   1:  PR[91,1] = PR[90,1] + 57.094;
   1:  PR[91,2] = PR[90,2] + 1.067;
   1:L PR[91] R[100]mm/sec CNT100;
   1:  PR[91,1] = PR[90,1] + 56.945;
   1:  PR[91,2] = PR[90,2] + -0.641;
   1:L PR[91] R[100]mm/sec CNT100;
   1:  PR[91,1] = PR[90,1] + 57.405;
   1:  PR[91,2] = PR[90,2] + -3.252;
   1:L PR[91] R[100]mm/sec CNT100;
   1:  PR[91,1] = PR[90,1] + 57.578;
   1:  PR[91,2] = PR[90,2] + -5.222;
   1:L PR[91] R[100]mm/sec CNT100;
   1:  PR[91,1] = PR[90,1] + 58.023;
   1:  PR[91,2] = PR[90,2] + -6.884;
   1:L PR[91] R[100]mm/sec CNT100;
   1:  PR[91,1] = PR[90,1] + 58.785;
   1:  PR[91,2] = PR[90,2] + -8.519;
   1:L PR[91] R[100]mm/sec CNT100;
   1:  PR[91,1] = PR[90,1] + 60.110;
   1:  PR[91,2] = PR[90,2] + -10.814;
   1:L PR[91] R[100]mm/sec CNT100;
   1:  PR[91,1] = PR[90,1] + 61.097;
   1:  PR[91,2] = PR[90,2] + -12.224;
   1:L PR[91] R[100]mm/sec CNT100;
   1:  PR[91,1] = PR[90,1] + 63.127;
   1:  PR[91,2] = PR[90,2] + -13.927;
   1:L PR[91] R[100]mm/sec CNT100;
   1:  PR[91,1] = PR[90,1] + 64.524;
   1:  PR[91,2] = PR[90,2] + -15.324;
   1:L PR[91] R[100]mm/sec CNT100;
   1:  PR[91,1] = PR[90,1] + 65.861;
   1:  PR[91,2] = PR[90,2] + -16.260;
   1:L PR[91] R[100]mm/sec CNT100;
   1:  PR[91,1] = PR[90,1] + 68.351;
   1:  PR[91,2] = PR[90,2] + -17.167;
   1:L PR[91] R[100]mm/sec CNT100;
   1:  PR[91,1] = PR[90,1] + 70.142;
   1:  PR[91,2] = PR[90,2] + -18.003;
   1:L PR[91] R[100]mm/sec CNT100;
   1:  PR[91,1] = PR[90,1] + 71.802;
   1:  PR[91,2] = PR[90,2] + -18.448;
   1:L PR[91] R[100]mm/sec CNT100;
   1:  PR[91,1] = PR[90,1] + 73.599;
   1:  PR[91,2] = PR[90,2] + -18.606;
   1:L PR[91] R[100]mm/sec CNT100;
   1:  PR[91,1] = PR[90,1] + 76.252;
   1:L PR[91] R[100]mm/sec CNT100;
   1:  PR[91,1] = PR[90,1] + 78.050;
   1:  PR[91,2] = PR[90,2] + -18.449;
   1:L PR[91] R[100]mm/sec CNT100;
   1:  PR[91,1] = PR[90,1] + 79.796;
   1:  PR[91,2] = PR[90,2] + -17.982;
   1:L PR[91] R[100]mm/sec CNT100;
   1:  PR[91,1] = PR[90,1] + 82.287;
   1:  PR[91,2] = PR[90,2] + -17.075;
   1:L PR[91] R[100]mm/sec CNT100;
   1:  PR[91,1] = PR[90,1] + 83.922;
   1:  PR[91,2] = PR[90,2] + -16.313;
   1:L PR[91] R[100]mm/sec CNT100;
   1:  PR[91,1] = PR[90,1] + 85.403;
   1:  PR[91,2] = PR[90,2] + -15.277;
   1:L PR[91] R[100]mm/sec CNT100;
   1:  PR[91,1] = PR[90,1] + 87.434;
   1:  PR[91,2] = PR[90,2] + -13.573;
   1:L PR[91] R[100]mm/sec CNT100;
   1:  PR[91,1] = PR[90,1] + 88.709;
   1:  PR[91,2] = PR[90,2] + -12.298;
   1:L PR[91] R[100]mm/sec CNT100;
   1:  PR[91,1] = PR[90,1] + 89.747;
   1:  PR[91,2] = PR[90,2] + -10.816;
   1:L PR[91] R[100]mm/sec CNT100;
   1:  PR[91,1] = PR[90,1] + 91.073;
   1:  PR[91,2] = PR[90,2] + -8.521;
   1:L PR[91] R[100]mm/sec CNT100;
   1:  PR[91,1] = PR[90,1] + 91.836;
   1:  PR[91,2] = PR[90,2] + -6.885;
   1:L PR[91] R[100]mm/sec CNT100;
   1:  PR[91,1] = PR[90,1] + 92.304;
   1:  PR[91,2] = PR[90,2] + -5.137;
   1:L PR[91] R[100]mm/sec CNT100;
   1:  PR[91,1] = PR[90,1] + 92.765;
   1:  PR[91,2] = PR[90,2] + -2.525;
   1:L PR[91] R[100]mm/sec CNT100;
   1:  PR[91,1] = PR[90,1] + 92.914;
   1:  PR[91,2] = PR[90,2] + -0.818;
   1:L PR[91] R[100]mm/sec CNT100;
   1:  PR[91,1] = PR[90,1] + 92.453;
   1:  PR[91,2] = PR[90,2] + 1.793;
   1:L PR[91] R[100]mm/sec CNT100;
   1:  PR[91,1] = PR[90,1] + 92.281;
   1:  PR[91,2] = PR[90,2] + 3.763;
   1:L PR[91] R[100]mm/sec CNT100;
   1:  PR[91,1] = PR[90,1] + 91.836;
   1:  PR[91,2] = PR[90,2] + 5.425;
   1:L PR[91] R[100]mm/sec CNT100;
   1:  PR[91,1] = PR[90,1] + 91.074;
   1:  PR[91,2] = PR[90,2] + 7.060;
   1:L PR[91] R[100]mm/sec CNT100;
   1:  PR[91,1] = PR[90,1] + 89.749;
   1:  PR[91,2] = PR[90,2] + 9.355;
   1:L PR[91] R[100]mm/sec CNT100;
   1:  PR[91,1] = PR[90,1] + 88.761;
   1:  PR[91,2] = PR[90,2] + 10.765;
   1:L PR[91] R[100]mm/sec CNT100TB   .50sec,CALL END_PUD;
   1:  PR[92] = PR[91];
   1:  PR[92,3] = PR[92,3] + 20;
   1:J PR[92] 10% FINE;
   1:  PR[91] = PR[90];
   1:  PR[91,1] = PR[90,1] + -91.940;
   1:  PR[91,2] = PR[90,2] + 5.505;
   1:  PR[91,3] = PR[90,3] + 6.695;
   1:  PR[92] = PR[91];
   1:  PR[92,3] = PR[92,3] + 20;
   1:J PR[92] 10% FINE;
   1:L PR[91] R[100]mm/sec CNT100;
   1:  CALL LASER_DRAHT_START;
   1:  PR[91,1] = PR[90,1] + -92.205;
   1:  PR[91,2] = PR[90,2] + 4.006;
   1:L PR[91] R[100]mm/sec CNT100;
   1:  PR[91,1] = PR[90,1] + -92.864;
   1:  PR[91,2] = PR[90,2] + 1.543;
   1:L PR[91] R[100]mm/sec CNT100;
   1:  PR[91,1] = PR[90,1] + -93.055;
   1:  PR[91,2] = PR[90,2] + -0.641;
   1:L PR[91] R[100]mm/sec CNT100;
   1:  PR[91,1] = PR[90,1] + -92.791;
   1:  PR[91,2] = PR[90,2] + -2.140;
   1:L PR[91] R[100]mm/sec CNT100;
   1:  PR[91,1] = PR[90,1] + -92.569;
   1:  PR[91,2] = PR[90,2] + -4.674;
   1:L PR[91] R[100]mm/sec CNT100;
   1:  PR[91,1] = PR[90,1] + -92.000;
   1:  PR[91,2] = PR[90,2] + -6.799;
   1:L PR[91] R[100]mm/sec CNT100;
   1:  PR[91,1] = PR[90,1] + -91.239;
   1:  PR[91,2] = PR[90,2] + -8.116;
   1:L PR[91] R[100]mm/sec CNT100;
   1:  PR[91,1] = PR[90,1] + -90.163;
   1:  PR[91,2] = PR[90,2] + -10.424;
   1:L PR[91] R[100]mm/sec CNT100;
   1:  PR[91,1] = PR[90,1] + -88.900;
   1:  PR[91,2] = PR[90,2] + -12.227;
   1:L PR[91] R[100]mm/sec CNT100;
   1:  PR[91,1] = PR[90,1] + -87.735;
   1:  PR[91,2] = PR[90,2] + -13.205;
   1:L PR[91] R[100]mm/sec CNT100;
   1:  PR[91,1] = PR[90,1] + -85.936;
   1:  PR[91,2] = PR[90,2] + -15.002;
   1:L PR[91] R[100]mm/sec CNT100;
   1:  PR[91,1] = PR[90,1] + -84.133;
   1:  PR[91,2] = PR[90,2] + -16.264;
   1:L PR[91] R[100]mm/sec CNT100;
   1:  PR[91,1] = PR[90,1] + -82.704;
   1:  PR[91,2] = PR[90,2] + -16.784;
   1:L PR[91] R[100]mm/sec CNT100;
   1:  PR[91,1] = PR[90,1] + -80.399;
   1:  PR[91,2] = PR[90,2] + -17.858;
   1:L PR[91] R[100]mm/sec CNT100;
   1:  PR[91,1] = PR[90,1] + -78.275;
   1:  PR[91,2] = PR[90,2] + -18.427;
   1:L PR[91] R[100]mm/sec CNT100;
   1:  PR[91,1] = PR[90,1] + -76.752;
   1:L PR[91] R[100]mm/sec CNT100;
   1:  PR[91,1] = PR[90,1] + -74.216;
   1:  PR[91,2] = PR[90,2] + -18.647;
   1:L PR[91] R[100]mm/sec CNT100;
   1:  PR[91,1] = PR[90,1] + -72.030;
   1:  PR[91,2] = PR[90,2] + -18.455;
   1:L PR[91] R[100]mm/sec CNT100;
   1:  PR[91,1] = PR[90,1] + -70.601;
   1:  PR[91,2] = PR[90,2] + -17.935;
   1:L PR[91] R[100]mm/sec CNT100;
   1:  PR[91,1] = PR[90,1] + -68.141;
   1:  PR[91,2] = PR[90,2] + -17.275;
   1:L PR[91] R[100]mm/sec CNT100;
   1:  PR[91,1] = PR[90,1] + -66.075;
   1:  PR[91,2] = PR[90,2] + -16.311;
   1:L PR[91] R[100]mm/sec CNT100;
   1:  PR[91,1] = PR[90,1] + -64.129;
   1:  PR[91,2] = PR[90,2] + -14.949;
   1:L PR[91] R[100]mm/sec CNT100;
   1:  PR[91,1] = PR[90,1] + -62.963;
   1:  PR[91,2] = PR[90,2] + -13.970;
   1:L PR[91] R[100]mm/sec CNT100;
   1:  PR[91,1] = PR[90,1] + -61.289;
   1:  PR[91,2] = PR[90,2] + -12.296;
   1:L PR[91] R[100]mm/sec CNT100;
   1:  PR[91,1] = PR[90,1] + -59.926;
   1:  PR[91,2] = PR[90,2] + -10.349;
   1:L PR[91] R[100]mm/sec CNT100;
   1:  PR[91,1] = PR[90,1] + -59.165;
   1:  PR[91,2] = PR[90,2] + -9.031;
   1:L PR[91] R[100]mm/sec CNT100;
   1:  PR[91,1] = PR[90,1] + -58.201;
   1:  PR[91,2] = PR[90,2] + -6.963;
   1:L PR[91] R[100]mm/sec CNT100;
   1:  PR[91,1] = PR[90,1] + -57.936;
   1:  PR[91,2] = PR[90,2] + -5.465;
   1:L PR[91] R[100]mm/sec CNT100;
   1:  PR[91,1] = PR[90,1] + -57.277;
   1:  PR[91,2] = PR[90,2] + -3.002;
   1:L PR[91] R[100]mm/sec CNT100;
   1:  PR[91,1] = PR[90,1] + -57.086;
   1:  PR[91,2] = PR[90,2] + -0.818;
   1:L PR[91] R[100]mm/sec CNT100;
   1:  PR[91,1] = PR[90,1] + -57.350;
   1:  PR[91,2] = PR[90,2] + 0.681;
   1:L PR[91] R[100]mm/sec CNT100;
   1:  PR[91,1] = PR[90,1] + -57.572;
   1:  PR[91,2] = PR[90,2] + 3.215;
   1:L PR[91] R[100]mm/sec CNT100;
   1:  PR[91,1] = PR[90,1] + -58.141;
   1:  PR[91,2] = PR[90,2] + 5.341;
   1:L PR[91] R[100]mm/sec CNT100;
   1:  PR[91,1] = PR[90,1] + -58.902;
   1:  PR[91,2] = PR[90,2] + 6.658;
   1:L PR[91] R[100]mm/sec CNT100;
   1:  PR[91,1] = PR[90,1] + -59.978;
   1:  PR[91,2] = PR[90,2] + 8.965;
   1:L PR[91] R[100]mm/sec CNT100;
   1:  PR[91,1] = PR[90,1] + -61.241;
   1:  PR[91,2] = PR[90,2] + 10.768;
   1:L PR[91] R[100]mm/sec CNT100;
   1:  PR[91,1] = PR[90,1] + -62.406;
   1:  PR[91,2] = PR[90,2] + 11.746;
   1:L PR[91] R[100]mm/sec CNT100;
   1:  PR[91,1] = PR[90,1] + -64.205;
   1:  PR[91,2] = PR[90,2] + 13.543;
   1:L PR[91] R[100]mm/sec CNT100;
   1:  PR[91,1] = PR[90,1] + -66.008;
   1:  PR[91,2] = PR[90,2] + 14.805;
   1:L PR[91] R[100]mm/sec CNT100;
   1:  PR[91,1] = PR[90,1] + -67.437;
   1:  PR[91,2] = PR[90,2] + 15.326;
   1:L PR[91] R[100]mm/sec CNT100;
   1:  PR[91,1] = PR[90,1] + -69.742;
   1:  PR[91,2] = PR[90,2] + 16.399;
   1:L PR[91] R[100]mm/sec CNT100;
   1:  PR[91,1] = PR[90,1] + -71.866;
   1:  PR[91,2] = PR[90,2] + 16.968;
   1:L PR[91] R[100]mm/sec CNT100;
   1:  PR[91,1] = PR[90,1] + -73.389;
   1:L PR[91] R[100]mm/sec CNT100;
   1:  PR[91,1] = PR[90,1] + -75.925;
   1:  PR[91,2] = PR[90,2] + 17.189;
   1:L PR[91] R[100]mm/sec CNT100;
   1:  PR[91,1] = PR[90,1] + -78.111;
   1:  PR[91,2] = PR[90,2] + 16.997;
   1:L PR[91] R[100]mm/sec CNT100;
   1:  PR[91,1] = PR[90,1] + -79.540;
   1:  PR[91,2] = PR[90,2] + 16.476;
   1:L PR[91] R[100]mm/sec CNT100;
   1:  PR[91,1] = PR[90,1] + -82.001;
   1:  PR[91,2] = PR[90,2] + 15.816;
   1:L PR[91] R[100]mm/sec CNT100;
   1:  PR[91,1] = PR[90,1] + -84.067;
   1:  PR[91,2] = PR[90,2] + 14.852;
   1:L PR[91] R[100]mm/sec CNT100;
   1:  PR[91,1] = PR[90,1] + -86.012;
   1:  PR[91,2] = PR[90,2] + 13.490;
   1:L PR[91] R[100]mm/sec CNT100;
   1:  PR[91,1] = PR[90,1] + -87.178;
   1:  PR[91,2] = PR[90,2] + 12.512;
   1:L PR[91] R[100]mm/sec CNT100;
   1:  PR[91,1] = PR[90,1] + -88.852;
   1:  PR[91,2] = PR[90,2] + 10.838;
   1:L PR[91] R[100]mm/sec CNT100;
   1:  PR[91,1] = PR[90,1] + -90.215;
   1:  PR[91,2] = PR[90,2] + 8.891;
   1:L PR[91] R[100]mm/sec CNT100;
   1:  PR[91,1] = PR[90,1] + -90.976;
   1:  PR[91,2] = PR[90,2] + 7.572;
   1:L PR[91] R[100]mm/sec CNT100;
   1:  PR[91,1] = PR[90,1] + -91.940;
   1:  PR[91,2] = PR[90,2] + 5.505;
   1:L PR[91] R[100]mm/sec CNT100TB   .50sec,CALL END_PUD;
   1:  PR[92] = PR[91];
   1:  PR[92,3] = PR[92,3] + 20;
   1:J PR[92] 10% FINE;
   1:  PR[91,1] = PR[90,1] + -42.791;
   1:  PR[91,2] = PR[90,2] + -2.140;
   1:  PR[92] = PR[91];
   1:  PR[92,3] = PR[92,3] + 20;
   1:J PR[92] 10% FINE;
   1:L PR[91] R[100]mm/sec CNT100;
   1:  CALL LASER_DRAHT_START;
   1:  PR[91,1] = PR[90,1] + -42.569;
   1:  PR[91,2] = PR[90,2] + -4.674;
   1:L PR[91] R[100]mm/sec CNT100;
   1:  PR[91,1] = PR[90,1] + -41.979;
